LIN {X 0,Y 256.069,Z 339.565,A -85,B 0,C 180,E1 -18517.403,E2 -18517.403} C_VEL
LIN {X 0,Y 256.173,Z 339.546,A -85,B 0,C 180,E1 -18520.779,E2 -18520.779} C_VEL
LIN {X 0,Y 256.276,Z 339.562,A -85,B 0,C 180,E1 -18524.084,E2 -18524.084} C_VEL
LIN {X 0,Y 256.286,Z 339.555,A -85,B 0,C 180,E1 -18528.933,E2 -18528.933} C_VEL
LIN {X 0,Y 256.491,Z 339.526,A -85,B 0,C 180,E1 -18532.126,E2 -18532.126} C_VEL
LIN {X 0,Y 256.447,Z 339.54,A -85,B 0,C 180,E1 -18536.858,E2 -18536.858} C_VEL
LIN {X 0,Y 256.694,Z 339.506,A -85,B 0,C 180,E1 -18538.431,E2 -18538.431} C_VEL
LIN {X 0,Y 256.692,Z 339.489,A -85,B 0,C 180,E1 -18541.569,E2 -18541.569} C_VEL
LIN {X 0,Y 256.437,Z 339.527,A -85,B 0,C 180,E1 -18546.594,E2 -18546.594} C_VEL
LIN {X 0,Y 256.423,Z 339.532,A -85,B 0,C 180,E1 -18549.465,E2 -18549.465} C_VEL
LIN {X 0,Y 256.231,Z 339.545,A -85,B 0,C 180,E1 -18554.292,E2 -18554.292} C_VEL
LIN {X 0,Y 256.173,Z 339.575,A -85,B 0,C 180,E1 -18557.565,E2 -18557.565} C_VEL
LIN {X 0,Y 256.133,Z 339.561,A -85,B 0,C 180,E1 -18561.108,E2 -18561.108} C_VEL
LIN {X 0,Y 256.078,Z 339.583,A -85,B 0,C 180,E1 -18565.088,E2 -18565.088} C_VEL
LIN {X 0,Y 256.072,Z 339.529,A -85,B 0,C 180,E1 -18568.57,E2 -18568.57} C_VEL
LIN {X 0,Y 256.066,Z 339.546,A -85,B 0,C 180,E1 -18571.7,E2 -18571.7} C_VEL
LIN {X 0,Y 256.076,Z 339.588,A -85,B 0,C 180,E1 -18575.194,E2 -18575.194} C_VEL
LIN {X 0,Y 256.062,Z 339.542,A -85,B 0,C 180,E1 -18579.144,E2 -18579.144} C_VEL
LIN {X 0,Y 256.02,Z 339.597,A -85,B 0,C 180,E1 -18583.336,E2 -18583.336} C_VEL
LIN {X 0,Y 256.031,Z 339.564,A -85,B 0,C 180,E1 -18587.829,E2 -18587.829} C_VEL
LIN {X 0,Y 256.064,Z 339.581,A -85,B 0,C 180,E1 -18590.857,E2 -18590.857} C_VEL
LIN {X 0,Y 256.078,Z 339.583,A -85,B 0,C 180,E1 -18594.807,E2 -18594.807} C_VEL
LIN {X 0,Y 256.112,Z 339.714,A -85,B 0,C 180,E1 -18598.125,E2 -18598.125} C_VEL
LIN {X 0,Y 256.299,Z 340.625,A -85,B 0,C 180,E1 -18598.413,E2 -18598.413} C_VEL
LIN {X 0,Y 265.977,Z 358.451,A -85,B 0,C 180,E1 -18600.315,E2 -18600.315} C_VEL
LIN {X 0,Y 273.395,Z 374.129,A -85,B 0,C 180,E1 -18601.697,E2 -18601.697} C_VEL
LIN {X 0,Y 273.811,Z 374.994,A -85,B 0,C 180,E1 -18601.771,E2 -18601.771} C_VEL
LIN {X 0,Y 272.891,Z 418.973,A -85,B 0,C 180,E1 -18602.963,E2 -18602.963} C_VEL
LIN {X 0,Y 272.46,Z 432.928,A -85,B 0,C 180,E1 -18603.563,E2 -18603.563} C_VEL
LIN {X 0,Y 271.747,Z 444.5,A -85,B 0,C 180,E1 -18604.331,E2 -18604.331} C_VEL
LIN {X 0,Y 270.545,Z 456.738,A -85,B 0,C 180,E1 -18605.441,E2 -18605.441} C_VEL
LIN {X 0,Y 269.175,Z 467,A -85,B 0,C 180,E1 -18606.638,E2 -18606.638} C_VEL
LIN {X 0,Y 267.356,Z 477.747,A -85,B 0,C 180,E1 -18608.204,E2 -18608.204} C_VEL
LIN {X 0,Y 265.658,Z 486.939,A -85,B 0,C 180,E1 -18609.885,E2 -18609.885} C_VEL
LIN {X 0,Y 264.051,Z 495.288,A -85,B 0,C 180,E1 -18611.776,E2 -18611.776} C_VEL
LIN {X 0,Y 262.199,Z 503.403,A -85,B 0,C 180,E1 -18614.054,E2 -18614.054} C_VEL
LIN {X 0,Y 260.462,Z 510.51,A -85,B 0,C 180,E1 -18616.578,E2 -18616.578} C_VEL
LIN {X 0,Y 259.237,Z 515.882,A -85,B 0,C 180,E1 -18619.061,E2 -18619.061} C_VEL
LIN {X 0,Y 258.088,Z 519.772,A -85,B 0,C 180,E1 -18621.387,E2 -18621.387} C_VEL
LIN {X 0,Y 257.177,Z 522.649,A -85,B 0,C 180,E1 -18623.725,E2 -18623.725} C_VEL
LIN {X 0,Y 257.015,Z 523.987,A -85,B 0,C 180,E1 -18625.295,E2 -18625.295} C_VEL
LIN {X 0,Y 256.72,Z 524.962,A -85,B 0,C 180,E1 -18626.861,E2 -18626.861} C_VEL
LIN {X 0,Y 256.704,Z 525.54,A -85,B 0,C 180,E1 -18628.431,E2 -18628.431} C_VEL
LIN {X 0,Y 256.664,Z 525.764,A -85,B 0,C 180,E1 -18630,E2 -18630} C_VEL
LIN {X 0,Y 256.704,Z 525.576,A -85,B 0,C 180,E1 -18631.569,E2 -18631.569} C_VEL
LIN {X 0,Y 256.719,Z 525.022,A -85,B 0,C 180,E1 -18633.139,E2 -18633.139} C_VEL
LIN {X 0,Y 257.009,Z 524.07,A -85,B 0,C 180,E1 -18634.706,E2 -18634.706} C_VEL
LIN {X 0,Y 257.163,Z 522.771,A -85,B 0,C 180,E1 -18636.276,E2 -18636.276} C_VEL
LIN {X 0,Y 258.081,Z 519.939,A -85,B 0,C 180,E1 -18638.614,E2 -18638.614} C_VEL
LIN {X 0,Y 259.211,Z 516.108,A -85,B 0,C 180,E1 -18640.94,E2 -18640.94} C_VEL
LIN {X 0,Y 260.376,Z 511.024,A -85,B 0,C 180,E1 -18643.342,E2 -18643.342} C_VEL
LIN {X 0,Y 262.21,Z 503.778,A -85,B 0,C 180,E1 -18645.946,E2 -18645.946} C_VEL
LIN {X 0,Y 264.037,Z 495.746,A -85,B 0,C 180,E1 -18648.225,E2 -18648.225} C_VEL
LIN {X 0,Y 265.659,Z 487.519,A -85,B 0,C 180,E1 -18650.115,E2 -18650.115} C_VEL
LIN {X 0,Y 267.297,Z 478.476,A -85,B 0,C 180,E1 -18651.801,E2 -18651.801} C_VEL
LIN {X 0,Y 269.348,Z 466.924,A -85,B 0,C 180,E1 -18653.483,E2 -18653.483} C_VEL
LIN {X 0,Y 270.868,Z 454.986,A -85,B 0,C 180,E1 -18654.859,E2 -18654.859} C_VEL
LIN {X 0,Y 272.101,Z 442.376,A -85,B 0,C 180,E1 -18655.932,E2 -18655.932} C_VEL
LIN {X 0,Y 272.774,Z 430.266,A -85,B 0,C 180,E1 -18656.684,E2 -18656.684} C_VEL
LIN {X 0,Y 272.92,Z 419.568,A -85,B 0,C 180,E1 -18657.142,E2 -18657.142} C_VEL
LIN {X 0,Y 273.881,Z 375.117,A -85,B 0,C 180,E1 -18658.347,E2 -18658.347} C_VEL
LIN {X 0,Y 266.772,Z 359.974,A -85,B 0,C 180,E1 -18659.671,E2 -18659.671} C_VEL
LIN {X 0,Y 259.254,Z 346.14,A -85,B 0,C 180,E1 -18661.101,E2 -18661.101} C_VEL
LIN {X 0,Y 256.306,Z 340.687,A -85,B 0,C 180,E1 -18661.719,E2 -18661.719} C_VEL
LIN {X 0,Y 256.095,Z 339.689,A -85,B 0,C 180,E1 -18662.04,E2 -18662.04} C_VEL
LIN {X 0,Y 256.077,Z 339.586,A -85,B 0,C 180,E1 -18665.193,E2 -18665.193} C_VEL
LIN {X 0,Y 256.041,Z 339.582,A -85,B 0,C 180,E1 -18669.147,E2 -18669.147} C_VEL
LIN {X 0,Y 256.001,Z 339.563,A -85,B 0,C 180,E1 -18673.339,E2 -18673.339} C_VEL
LIN {X 0,Y 256.031,Z 339.586,A -85,B 0,C 180,E1 -18677.828,E2 -18677.828} C_VEL
LIN {X 0,Y 256.062,Z 339.543,A -85,B 0,C 180,E1 -18680.856,E2 -18680.856} C_VEL
LIN {X 0,Y 256.076,Z 339.587,A -85,B 0,C 180,E1 -18684.806,E2 -18684.806} C_VEL
LIN {X 0,Y 256.074,Z 339.541,A -85,B 0,C 180,E1 -18688.57,E2 -18688.57} C_VEL
LIN {X 0,Y 256.073,Z 339.538,A -85,B 0,C 180,E1 -18692.188,E2 -18692.188} C_VEL
LIN {X 0,Y 256.081,Z 339.586,A -85,B 0,C 180,E1 -18695.69,E2 -18695.69} C_VEL
LIN {X 0,Y 256.117,Z 339.563,A -85,B 0,C 180,E1 -18699.1,E2 -18699.1} C_VEL
LIN {X 0,Y 256.226,Z 339.555,A -85,B 0,C 180,E1 -18704.08,E2 -18704.08} C_VEL
LIN {X 0,Y 256.286,Z 339.56,A -85,B 0,C 180,E1 -18708.933,E2 -18708.933} C_VEL
LIN {X 0,Y 256.462,Z 339.518,A -85,B 0,C 180,E1 -18712.125,E2 -18712.125} C_VEL
LIN {X 0,Y 256.449,Z 339.535,A -85,B 0,C 180,E1 -18716.858,E2 -18716.858} C_VEL
LIN {X 0,Y 256.691,Z 339.489,A -85,B 0,C 180,E1 -18718.431,E2 -18718.431} C_VEL
LIN {X 0,Y 256.637,Z 339.511,A -85,B 0,C 180,E1 -18721.842,E2 -18721.842} C_VEL
LIN {X 0,Y 256.452,Z 339.518,A -85,B 0,C 180,E1 -18726.293,E2 -18726.293} C_VEL
LIN {X 0,Y 256.424,Z 339.535,A -85,B 0,C 180,E1 -18728.703,E2 -18728.703} C_VEL
LIN {X 0,Y 255.723,Z 339.631,A -85,B 0,C 180,E1 -18730.013,E2 -18730.013} C_VEL
LIN {X 0,Y 252.772,Z 339.993,A -85,B 0,C 180,E1 -18732.144,E2 -18732.144} C_VEL
LIN {X 0,Y 250.284,Z 340.298,A -85,B 0,C 180,E1 -18733.88,E2 -18733.88} C_VEL
LIN {X 0,Y 249.236,Z 340.437,A -85,B 0,C 180,E1 -18735.229,E2 -18735.229} C_VEL
LIN {X 0,Y 249.16,Z 340.442,A -85,B 0,C 180,E1 -18735.686,E2 -18735.686} C_VEL
LIN {X 0,Y 249.08,Z 340.421,A -85,B 0,C 180,E1 -18739.791,E2 -18739.791} C_VEL
LIN {X 0,Y 249.039,Z 340.452,A -85,B 0,C 180,E1 -18743.271,E2 -18743.271} C_VEL
LIN {X 0,Y 249.02,Z 340.448,A -85,B 0,C 180,E1 -18746.844,E2 -18746.844} C_VEL
LIN {X 0,Y 248.998,Z 340.46,A -85,B 0,C 180,E1 -18750.534,E2 -18750.534} C_VEL
LIN {X 0,Y 249.04,Z 340.444,A -85,B 0,C 180,E1 -18755.077,E2 -18755.077} C_VEL
LIN {X 0,Y 249.02,Z 340.455,A -85,B 0,C 180,E1 -18758.382,E2 -18758.382} C_VEL
LIN {X 0,Y 248.98,Z 340.447,A -85,B 0,C 180,E1 -18762.786,E2 -18762.786} C_VEL
LIN {X 0,Y 248.985,Z 340.61,A -85,B 0,C 180,E1 -18765.118,E2 -18765.118} C_VEL
LIN {X 0,Y 252.25,Z 352.179,A -85,B 0,C 180,E1 -18769.37,E2 -18769.37} C_VEL
LIN {X 0,Y 254.64,Z 361.802,A -85,B 0,C 180,E1 -18772.614,E2 -18772.614} C_VEL
LIN {X 0,Y 256.671,Z 371.259,A -85,B 0,C 180,E1 -18775.613,E2 -18775.613} C_VEL
LIN {X 0,Y 257.459,Z 376.644,A -85,B 0,C 180,E1 -18777.232,E2 -18777.232} C_VEL
LIN {X 0,Y 257.14,Z 378.887,A -85,B 0,C 180,E1 -18777.719,E2 -18777.719} C_VEL
LIN {X 0,Y 260.773,Z 406.312,A -85,B 0,C 180,E1 -18779.087,E2 -18779.087} C_VEL
LIN {X 0,Y 263.817,Z 435.444,A -85,B 0,C 180,E1 -18780.357,E2 -18780.357} C_VEL
LIN {X 0,Y 265.192,Z 455.664,A -85,B 0,C 180,E1 -18781.128,E2 -18781.128} C_VEL
LIN {X 0,Y 263.991,Z 490.905,A -85,B 0,C 180,E1 -18782.108,E2 -18782.108} C_VEL
LIN {X 0,Y 262.825,Z 504.718,A -85,B 0,C 180,E1 -18782.791,E2 -18782.791} C_VEL
LIN {X 0,Y 261.078,Z 517.612,A -85,B 0,C 180,E1 -18783.738,E2 -18783.738} C_VEL
LIN {X 0,Y 259.146,Z 529.368,A -85,B 0,C 180,E1 -18784.929,E2 -18784.929} C_VEL
LIN {X 0,Y 256.812,Z 540.726,A -85,B 0,C 180,E1 -18786.408,E2 -18786.408} C_VEL
LIN {X 0,Y 254.578,Z 551.008,A -85,B 0,C 180,E1 -18788.119,E2 -18788.119} C_VEL
LIN {X 0,Y 252.455,Z 560.299,A -85,B 0,C 180,E1 -18790.061,E2 -18790.061} C_VEL
LIN {X 0,Y 250.616,Z 569.039,A -85,B 0,C 180,E1 -18792.34,E2 -18792.34} C_VEL
LIN {X 0,Y 249.503,Z 574.497,A -85,B 0,C 180,E1 -18794.06,E2 -18794.06} C_VEL
LIN {X 0,Y 248.311,Z 581.828,A -85,B 0,C 180,E1 -18796.914,E2 -18796.914} C_VEL
LIN {X 0,Y 247.795,Z 586.756,A -85,B 0,C 180,E1 -18799.377,E2 -18799.377} C_VEL
LIN {X 0,Y 247.778,Z 590.581,A -85,B 0,C 180,E1 -18801.847,E2 -18801.847} C_VEL
LIN {X 0,Y 247.949,Z 592.578,A -85,B 0,C 180,E1 -18803.49,E2 -18803.49} C_VEL
LIN {X 0,Y 248.237,Z 594.099,A -85,B 0,C 180,E1 -18805.128,E2 -18805.128} C_VEL
LIN {X 0,Y 248.493,Z 595.191,A -85,B 0,C 180,E1 -18806.757,E2 -18806.757} C_VEL
LIN {X 0,Y 248.804,Z 595.878,A -85,B 0,C 180,E1 -18808.381,E2 -18808.381} C_VEL
LIN {X 0,Y 249.239,Z 596.163,A -85,B 0,C 180,E1 -18810,E2 -18810} C_VEL
LIN {X 0,Y 248.809,Z 595.869,A -85,B 0,C 180,E1 -18811.619,E2 -18811.619} C_VEL
LIN {X 0,Y 248.504,Z 595.178,A -85,B 0,C 180,E1 -18813.242,E2 -18813.242} C_VEL
LIN {X 0,Y 248.257,Z 594.082,A -85,B 0,C 180,E1 -18814.872,E2 -18814.872} C_VEL
LIN {X 0,Y 247.899,Z 591.823,A -85,B 0,C 180,E1 -18817.132,E2 -18817.132} C_VEL
LIN {X 0,Y 247.761,Z 588.091,A -85,B 0,C 180,E1 -18819.799,E2 -18819.799} C_VEL
LIN {X 0,Y 248.096,Z 583.525,A -85,B 0,C 180,E1 -18822.266,E2 -18822.266} C_VEL
LIN {X 0,Y 248.876,Z 577.769,A -85,B 0,C 180,E1 -18824.723,E2 -18824.723} C_VEL
LIN {X 0,Y 249.858,Z 571.762,A -85,B 0,C 180,E1 -18826.805,E2 -18826.805} C_VEL
LIN {X 0,Y 251.413,Z 564.965,A -85,B 0,C 180,E1 -18828.752,E2 -18828.752} C_VEL
LIN {X 0,Y 253.248,Z 556.625,A -85,B 0,C 180,E1 -18830.721,E2 -18830.721} C_VEL
LIN {X 0,Y 255.584,Z 546.518,A -85,B 0,C 180,E1 -18832.641,E2 -18832.641} C_VEL
LIN {X 0,Y 257.668,Z 536.556,A -85,B 0,C 180,E1 -18834.15,E2 -18834.15} C_VEL
LIN {X 0,Y 260.045,Z 523.989,A -85,B 0,C 180,E1 -18835.621,E2 -18835.621} C_VEL
LIN {X 0,Y 261.894,Z 511.65,A -85,B 0,C 180,E1 -18836.71,E2 -18836.71} C_VEL
LIN {X 0,Y 263.306,Z 498.554,A -85,B 0,C 180,E1 -18837.526,E2 -18837.526} C_VEL
LIN {X 0,Y 264.182,Z 485.189,A -85,B 0,C 180,E1 -18838.054,E2 -18838.054} C_VEL
LIN {X 0,Y 265.101,Z 453.13,A -85,B 0,C 180,E1 -18838.919,E2 -18838.919} C_VEL
LIN {X 0,Y 262.594,Z 423.589,A -85,B 0,C 180,E1 -18840.111,E2 -18840.111} C_VEL
LIN {X 0,Y 259.354,Z 395.566,A -85,B 0,C 180,E1 -18841.387,E2 -18841.387} C_VEL
LIN {X 0,Y 257.067,Z 378.809,A -85,B 0,C 180,E1 -18842.247,E2 -18842.247} C_VEL
LIN {X 0,Y 257.402,Z 375.362,A -85,B 0,C 180,E1 -18843.097,E2 -18843.097} C_VEL
LIN {X 0,Y 255.441,Z 365.273,A -85,B 0,C 180,E1 -18846.216,E2 -18846.216} C_VEL
LIN {X 0,Y 252.585,Z 353.374,A -85,B 0,C 180,E1 -18850.154,E2 -18850.154} C_VEL
LIN {X 0,Y 249.584,Z 342.552,A -85,B 0,C 180,E1 -18854.06,E2 -18854.06} C_VEL
LIN {X 0,Y 248.977,Z 340.558,A -85,B 0,C 180,E1 -18854.884,E2 -18854.884} C_VEL
LIN {X 0,Y 248.99,Z 340.452,A -85,B 0,C 180,E1 -18857.357,E2 -18857.357} C_VEL
LIN {X 0,Y 249.04,Z 340.389,A -85,B 0,C 180,E1 -18862.2,E2 -18862.2} C_VEL
LIN {X 0,Y 249.039,Z 340.419,A -85,B 0,C 180,E1 -18865.639,E2 -18865.639} C_VEL
LIN {X 0,Y 248.998,Z 340.459,A -85,B 0,C 180,E1 -18869.466,E2 -18869.466} C_VEL
LIN {X 0,Y 249.02,Z 340.45,A -85,B 0,C 180,E1 -18873.156,E2 -18873.156} C_VEL
LIN {X 0,Y 249.04,Z 340.451,A -85,B 0,C 180,E1 -18876.729,E2 -18876.729} C_VEL
LIN {X 0,Y 249.094,Z 340.42,A -85,B 0,C 180,E1 -18880.21,E2 -18880.21} C_VEL
LIN {X 0,Y 249.22,Z 340.442,A -85,B 0,C 180,E1 -18883.62,E2 -18883.62} C_VEL
LIN {X 0,Y 249.23,Z 340.43,A -85,B 0,C 180,E1 -18888.616,E2 -18888.616} C_VEL
LIN {X 0,Y 249.434,Z 340.406,A -85,B 0,C 180,E1 -18891.901,E2 -18891.901} C_VEL
LIN {X 0,Y 249.259,Z 340.423,A -85,B 0,C 180,E1 -18895.148,E2 -18895.148} C_VEL
LIN {X 0,Y 249.655,Z 340.383,A -85,B 0,C 180,E1 -18898.387,E2 -18898.387} C_VEL
LIN {X 0,Y 249.653,Z 340.366,A -85,B 0,C 180,E1 -18901.613,E2 -18901.613} C_VEL
LIN {X 0,Y 249.414,Z 340.401,A -85,B 0,C 180,E1 -18906.573,E2 -18906.573} C_VEL
LIN {X 0,Y 249.339,Z 340.416,A -85,B 0,C 180,E1 -18909.737,E2 -18909.737} C_VEL
LIN {X 0,Y 249.174,Z 340.423,A -85,B 0,C 180,E1 -18914.705,E2 -18914.705} C_VEL
LIN {X 0,Y 249.108,Z 340.454,A -85,B 0,C 180,E1 -18918.08,E2 -18918.08} C_VEL
LIN {X 0,Y 249.073,Z 340.441,A -85,B 0,C 180,E1 -18921.52,E2 -18921.52} C_VEL
LIN {X 0,Y 249.039,Z 340.455,A -85,B 0,C 180,E1 -18925.44,E2 -18925.44} C_VEL
LIN {X 0,Y 249.02,Z 340.403,A -85,B 0,C 180,E1 -18928.969,E2 -18928.969} C_VEL
LIN {X 0,Y 249.022,Z 340.438,A -85,B 0,C 180,E1 -18932.427,E2 -18932.427} C_VEL
LIN {X 0,Y 249.01,Z 340.454,A -85,B 0,C 180,E1 -18936.349,E2 -18936.349} C_VEL
LIN {X 0,Y 248.976,Z 340.432,A -85,B 0,C 180,E1 -18940.484,E2 -18940.484} C_VEL
LIN {X 0,Y 248.96,Z 340.457,A -85,B 0,C 180,E1 -18944.889,E2 -18944.889} C_VEL
LIN {X 0,Y 248.977,Z 340.438,A -85,B 0,C 180,E1 -18947.355,E2 -18947.355} C_VEL
LIN {X 0,Y 249.017,Z 340.447,A -85,B 0,C 180,E1 -18951.619,E2 -18951.619} C_VEL
LIN {X 0,Y 249.042,Z 340.46,A -85,B 0,C 180,E1 -18955.64,E2 -18955.64} C_VEL
LIN {X 0,Y 249.084,Z 340.699,A -85,B 0,C 180,E1 -18957.164,E2 -18957.164} C_VEL
LIN {X 0,Y 249.404,Z 341.93,A -85,B 0,C 180,E1 -18957.457,E2 -18957.457} C_VEL
LIN {X 0,Y 258.456,Z 358.147,A -85,B 0,C 180,E1 -18959.31,E2 -18959.31} C_VEL
LIN {X 0,Y 265.998,Z 373.461,A -85,B 0,C 180,E1 -18960.778,E2 -18960.778} C_VEL
LIN {X 0,Y 267.575,Z 377.081,A -85,B 0,C 180,E1 -18961.084,E2 -18961.084} C_VEL
LIN {X 0,Y 266.644,Z 419.863,A -85,B 0,C 180,E1 -18962.272,E2 -18962.272} C_VEL
LIN {X 0,Y 266.201,Z 433.521,A -85,B 0,C 180,E1 -18962.868,E2 -18962.868} C_VEL
LIN {X 0,Y 265.425,Z 445.487,A -85,B 0,C 180,E1 -18963.673,E2 -18963.673} C_VEL
LIN {X 0,Y 264.169,Z 457.722,A -85,B 0,C 180,E1 -18964.808,E2 -18964.808} C_VEL
LIN {X 0,Y 262.738,Z 467.983,A -85,B 0,C 180,E1 -18966.03,E2 -18966.03} C_VEL
LIN {X 0,Y 260.844,Z 478.729,A -85,B 0,C 180,E1 -18967.631,E2 -18967.631} C_VEL
LIN {X 0,Y 259.069,Z 487.921,A -85,B 0,C 180,E1 -18969.35,E2 -18969.35} C_VEL
LIN {X 0,Y 257.384,Z 496.268,A -85,B 0,C 180,E1 -18971.287,E2 -18971.287} C_VEL
LIN {X 0,Y 255.448,Z 504.383,A -85,B 0,C 180,E1 -18973.621,E2 -18973.621} C_VEL
LIN {X 0,Y 253.631,Z 511.49,A -85,B 0,C 180,E1 -18976.21,E2 -18976.21} C_VEL
LIN {X 0,Y 252.34,Z 516.861,A -85,B 0,C 180,E1 -18978.758,E2 -18978.758} C_VEL
LIN {X 0,Y 251.142,Z 520.751,A -85,B 0,C 180,E1 -18981.146,E2 -18981.146} C_VEL
LIN {X 0,Y 250.189,Z 523.628,A -85,B 0,C 180,E1 -18983.549,E2 -18983.549} C_VEL
LIN {X 0,Y 250.01,Z 524.965,A -85,B 0,C 180,E1 -18985.162,E2 -18985.162} C_VEL
LIN {X 0,Y 249.703,Z 525.94,A -85,B 0,C 180,E1 -18986.773,E2 -18986.773} C_VEL
LIN {X 0,Y 249.679,Z 526.518,A -85,B 0,C 180,E1 -18988.387,E2 -18988.387} C_VEL
LIN {X 0,Y 249.636,Z 526.742,A -85,B 0,C 180,E1 -18990,E2 -18990} C_VEL
LIN {X 0,Y 249.679,Z 526.554,A -85,B 0,C 180,E1 -18991.613,E2 -18991.613} C_VEL
LIN {X 0,Y 249.702,Z 525.999,A -85,B 0,C 180,E1 -18993.227,E2 -18993.227} C_VEL
LIN {X 0,Y 250.004,Z 525.048,A -85,B 0,C 180,E1 -18994.838,E2 -18994.838} C_VEL
LIN {X 0,Y 250.174,Z 523.749,A -85,B 0,C 180,E1 -18996.452,E2 -18996.452} C_VEL
LIN {X 0,Y 251.135,Z 520.916,A -85,B 0,C 180,E1 -18998.854,E2 -18998.854} C_VEL
LIN {X 0,Y 252.315,Z 517.085,A -85,B 0,C 180,E1 -19001.243,E2 -19001.243} C_VEL
LIN {X 0,Y 253.543,Z 512,A -85,B 0,C 180,E1 -19003.709,E2 -19003.709} C_VEL
LIN {X 0,Y 255.459,Z 504.754,A -85,B 0,C 180,E1 -19006.379,E2 -19006.379} C_VEL
LIN {X 0,Y 257.371,Z 496.722,A -85,B 0,C 180,E1 -19008.714,E2 -19008.714} C_VEL
LIN {X 0,Y 259.069,Z 488.494,A -85,B 0,C 180,E1 -19010.65,E2 -19010.65} C_VEL
LIN {X 0,Y 260.785,Z 479.451,A -85,B 0,C 180,E1 -19012.374,E2 -19012.374} C_VEL
LIN {X 0,Y 262.729,Z 468.921,A -85,B 0,C 180,E1 -19013.96,E2 -19013.96} C_VEL
LIN {X 0,Y 264.342,Z 457.235,A -85,B 0,C 180,E1 -19015.364,E2 -19015.364} C_VEL
LIN {X 0,Y 265.643,Z 445.757,A -85,B 0,C 180,E1 -19016.41,E2 -19016.41} C_VEL
LIN {X 0,Y 266.365,Z 433.594,A -85,B 0,C 180,E1 -19017.241,E2 -19017.241} C_VEL
LIN {X 0,Y 266.676,Z 420.237,A -85,B 0,C 180,E1 -19017.843,E2 -19017.843} C_VEL
LIN {X 0,Y 267.652,Z 377.15,A -85,B 0,C 180,E1 -19019.037,E2 -19019.037} C_VEL
LIN {X 0,Y 260.711,Z 362.373,A -85,B 0,C 180,E1 -19020.387,E2 -19020.387} C_VEL
LIN {X 0,Y 252.472,Z 347.365,A -85,B 0,C 180,E1 -19022.029,E2 -19022.029} C_VEL
LIN {X 0,Y 249.294,Z 341.581,A -85,B 0,C 180,E1 -19022.729,E2 -19022.729} C_VEL
LIN {X 0,Y 249.048,Z 340.566,A -85,B 0,C 180,E1 -19023.087,E2 -19023.087} C_VEL
LIN {X 0,Y 249.01,Z 340.448,A -85,B 0,C 180,E1 -19026.348,E2 -19026.348} C_VEL
LIN {X 0,Y 248.97,Z 340.471,A -85,B 0,C 180,E1 -19030.484,E2 -19030.484} C_VEL
LIN {X 0,Y 248.96,Z 340.452,A -85,B 0,C 180,E1 -19034.888,E2 -19034.888} C_VEL
LIN {X 0,Y 248.977,Z 340.472,A -85,B 0,C 180,E1 -19037.354,E2 -19037.354} C_VEL
LIN {X 0,Y 249.041,Z 340.424,A -85,B 0,C 180,E1 -19042.2,E2 -19042.2} C_VEL
LIN {X 0,Y 249.04,Z 340.463,A -85,B 0,C 180,E1 -19045.639,E2 -19045.639} C_VEL
LIN {X 0,Y 248.99,Z 340.409,A -85,B 0,C 180,E1 -19049.464,E2 -19049.464} C_VEL
LIN {X 0,Y 249.009,Z 340.436,A -85,B 0,C 180,E1 -19053.155,E2 -19053.155} C_VEL
LIN {X 0,Y 249.002,Z 340.466,A -85,B 0,C 180,E1 -19056.725,E2 -19056.725} C_VEL
LIN {X 0,Y 249.052,Z 340.449,A -85,B 0,C 180,E1 -19060.207,E2 -19060.207} C_VEL
LIN {X 0,Y 249.154,Z 340.442,A -85,B 0,C 180,E1 -19063.616,E2 -19063.616} C_VEL
LIN {X 0,Y 249.229,Z 340.441,A -85,B 0,C 180,E1 -19068.615,E2 -19068.615} C_VEL
LIN {X 0,Y 249.412,Z 340.396,A -85,B 0,C 180,E1 -19071.9,E2 -19071.9} C_VEL
LIN {X 0,Y 249.26,Z 340.436,A -85,B 0,C 180,E1 -19075.148,E2 -19075.148} C_VEL
LIN {X 0,Y 249.653,Z 340.366,A -85,B 0,C 180,E1 -19078.387,E2 -19078.387} C_VEL
LIN {X 0,Y 249.655,Z 340.382,A -85,B 0,C 180,E1 -19081.613,E2 -19081.613} C_VEL
LIN {X 0,Y 249.423,Z 340.394,A -85,B 0,C 180,E1 -19086.471,E2 -19086.471} C_VEL
LIN {X 0,Y 249.339,Z 340.425,A -85,B 0,C 180,E1 -19089.737,E2 -19089.737} C_VEL
LIN {X 0,Y 249.177,Z 340.439,A -85,B 0,C 180,E1 -19094.705,E2 -19094.705} C_VEL
LIN {X 0,Y 249.16,Z 340.442,A -85,B 0,C 180,E1 -19095.686,E2 -19095.686} C_VEL
LIN {X 0,Y 248.504,Z 340.527,A -85,B 0,C 180,E1 -19097.035,E2 -19097.035} C_VEL
LIN {X 0,Y 245.605,Z 340.872,A -85,B 0,C 180,E1 -19099.233,E2 -19099.233} C_VEL
LIN {X 0,Y 243.125,Z 341.169,A -85,B 0,C 180,E1 -19101.023,E2 -19101.023} C_VEL
LIN {X 0,Y 242.058,Z 341.307,A -85,B 0,C 180,E1 -19102.414,E2 -19102.414} C_VEL
LIN {X 0,Y 241.971,Z 341.321,A -85,B 0,C 180,E1 -19102.886,E2 -19102.886} C_VEL
LIN {X 0,Y 241.988,Z 341.337,A -85,B 0,C 180,E1 -19105.826,E2 -19105.826} C_VEL
LIN {X 0,Y 241.965,Z 341.322,A -85,B 0,C 180,E1 -19109.589,E2 -19109.589} C_VEL
LIN {X 0,Y 241.976,Z 341.327,A -85,B 0,C 180,E1 -19113.493,E2 -19113.493} C_VEL
LIN {X 0,Y 241.981,Z 341.341,A -85,B 0,C 180,E1 -19117.584,E2 -19117.584} C_VEL
LIN {X 0,Y 241.915,Z 341.346,A -85,B 0,C 180,E1 -19121.927,E2 -19121.927} C_VEL
LIN {X 0,Y 241.93,Z 341.545,A -85,B 0,C 180,E1 -19124.202,E2 -19124.202} C_VEL
LIN {X 0,Y 244.942,Z 352.046,A -85,B 0,C 180,E1 -19128.246,E2 -19128.246} C_VEL
LIN {X 0,Y 247.415,Z 361.774,A -85,B 0,C 180,E1 -19131.687,E2 -19131.687} C_VEL
LIN {X 0,Y 249.909,Z 373.223,A -85,B 0,C 180,E1 -19135.462,E2 -19135.462} C_VEL
LIN {X 0,Y 250.67,Z 377.47,A -85,B 0,C 180,E1 -19136.741,E2 -19136.741} C_VEL
LIN {X 0,Y 252.007,Z 387.42,A -85,B 0,C 180,E1 -19137.314,E2 -19137.314} C_VEL
LIN {X 0,Y 254.816,Z 408.963,A -85,B 0,C 180,E1 -19138.397,E2 -19138.397} C_VEL
LIN {X 0,Y 257.963,Z 440.471,A -85,B 0,C 180,E1 -19139.8,E2 -19139.8} C_VEL
LIN {X 0,Y 258.942,Z 455.77,A -85,B 0,C 180,E1 -19140.396,E2 -19140.396} C_VEL
LIN {X 0,Y 257.731,Z 489.933,A -85,B 0,C 180,E1 -19141.369,E2 -19141.369} C_VEL
LIN {X 0,Y 256.53,Z 503.249,A -85,B 0,C 180,E1 -19142.031,E2 -19142.031} C_VEL
LIN {X 0,Y 254.926,Z 515.618,A -85,B 0,C 180,E1 -19142.943,E2 -19142.943} C_VEL
LIN {X 0,Y 253.049,Z 526.794,A -85,B 0,C 180,E1 -19144.06,E2 -19144.06} C_VEL
LIN {X 0,Y 250.607,Z 538.439,A -85,B 0,C 180,E1 -19145.566,E2 -19145.566} C_VEL
LIN {X 0,Y 248.198,Z 548.961,A -85,B 0,C 180,E1 -19147.307,E2 -19147.307} C_VEL
LIN {X 0,Y 246.186,Z 557.607,A -85,B 0,C 180,E1 -19149.094,E2 -19149.094} C_VEL
LIN {X 0,Y 244.331,Z 565.623,A -85,B 0,C 180,E1 -19151.12,E2 -19151.12} C_VEL
LIN {X 0,Y 242.537,Z 573.489,A -85,B 0,C 180,E1 -19153.589,E2 -19153.589} C_VEL
LIN {X 0,Y 241.339,Z 580.832,A -85,B 0,C 180,E1 -19156.528,E2 -19156.528} C_VEL
LIN {X 0,Y 240.763,Z 585.761,A -85,B 0,C 180,E1 -19159.063,E2 -19159.063} C_VEL
LIN {X 0,Y 240.708,Z 589.587,A -85,B 0,C 180,E1 -19161.606,E2 -19161.606} C_VEL
LIN {X 0,Y 240.856,Z 591.585,A -85,B 0,C 180,E1 -19163.297,E2 -19163.297} C_VEL
LIN {X 0,Y 241.145,Z 593.109,A -85,B 0,C 180,E1 -19164.984,E2 -19164.984} C_VEL
LIN {X 0,Y 241.432,Z 594.207,A -85,B 0,C 180,E1 -19166.662,E2 -19166.662} C_VEL
LIN {X 0,Y 241.741,Z 594.895,A -85,B 0,C 180,E1 -19168.334,E2 -19168.334} C_VEL
LIN {X 0,Y 242.198,Z 595.183,A -85,B 0,C 180,E1 -19170,E2 -19170} C_VEL
LIN {X 0,Y 241.443,Z 594.194,A -85,B 0,C 180,E1 -19173.337,E2 -19173.337} C_VEL
LIN {X 0,Y 241.166,Z 593.091,A -85,B 0,C 180,E1 -19175.015,E2 -19175.015} C_VEL
LIN {X 0,Y 240.823,Z 591.053,A -85,B 0,C 180,E1 -19177.146,E2 -19177.146} C_VEL
LIN {X 0,Y 240.686,Z 587.091,A -85,B 0,C 180,E1 -19180.09,E2 -19180.09} C_VEL
LIN {X 0,Y 241.087,Z 582.525,A -85,B 0,C 180,E1 -19182.629,E2 -19182.629} C_VEL
LIN {X 0,Y 241.954,Z 576.771,A -85,B 0,C 180,E1 -19185.154,E2 -19185.154} C_VEL
LIN {X 0,Y 242.857,Z 571.45,A -85,B 0,C 180,E1 -19187.069,E2 -19187.069} C_VEL
LIN {X 0,Y 244.631,Z 563.965,A -85,B 0,C 180,E1 -19189.292,E2 -19189.292} C_VEL
LIN {X 0,Y 246.571,Z 555.627,A -85,B 0,C 180,E1 -19191.31,E2 -19191.31} C_VEL
LIN {X 0,Y 248.956,Z 545.513,A -85,B 0,C 180,E1 -19193.279,E2 -19193.279} C_VEL
LIN {X 0,Y 251.479,Z 534.124,A -85,B 0,C 180,E1 -19195.004,E2 -19195.004} C_VEL
LIN {X 0,Y 253.659,Z 522.996,A -85,B 0,C 180,E1 -19196.314,E2 -19196.314} C_VEL
LIN {X 0,Y 255.581,Z 510.656,A -85,B 0,C 180,E1 -19197.425,E2 -19197.425} C_VEL
LIN {X 0,Y 257.023,Z 497.964,A -85,B 0,C 180,E1 -19198.234,E2 -19198.234} C_VEL
LIN {X 0,Y 257.922,Z 484.494,A -85,B 0,C 180,E1 -19198.786,E2 -19198.786} C_VEL
LIN {X 0,Y 258.862,Z 453.924,A -85,B 0,C 180,E1 -19199.628,E2 -19199.628} C_VEL
LIN {X 0,Y 256.159,Z 421.803,A -85,B 0,C 180,E1 -19200.972,E2 -19200.972} C_VEL
LIN {X 0,Y 252.598,Z 391.455,A -85,B 0,C 180,E1 -19202.424,E2 -19202.424} C_VEL
LIN {X 0,Y 250.59,Z 377.511,A -85,B 0,C 180,E1 -19203.216,E2 -19203.216} C_VEL
LIN {X 0,Y 249.442,Z 371.008,A -85,B 0,C 180,E1 -19205.207,E2 -19205.207} C_VEL
LIN {X 0,Y 247.386,Z 361.581,A -85,B 0,C 180,E1 -19208.327,E2 -19208.327} C_VEL
LIN {X 0,Y 244.508,Z 350.507,A -85,B 0,C 180,E1 -19212.256,E2 -19212.256} C_VEL
LIN {X 0,Y 241.923,Z 341.476,A -85,B 0,C 180,E1 -19215.796,E2 -19215.796} C_VEL
LIN {X 0,Y 241.939,Z 341.302,A -85,B 0,C 180,E1 -19220.277,E2 -19220.277} C_VEL
LIN {X 0,Y 241.97,Z 341.276,A -85,B 0,C 180,E1 -19224.486,E2 -19224.486} C_VEL
LIN {X 0,Y 241.95,Z 341.347,A -85,B 0,C 180,E1 -19228.476,E2 -19228.476} C_VEL
LIN {X 0,Y 241.958,Z 341.319,A -85,B 0,C 180,E1 -19232.306,E2 -19232.306} C_VEL
LIN {X 0,Y 242.005,Z 341.336,A -85,B 0,C 180,E1 -19236.01,E2 -19236.01} C_VEL
LIN {X 0,Y 242.025,Z 341.297,A -85,B 0,C 180,E1 -19239.607,E2 -19239.607} C_VEL
LIN {X 0,Y 242.16,Z 341.319,A -85,B 0,C 180,E1 -19243.278,E2 -19243.278} C_VEL
LIN {X 0,Y 242.165,Z 341.305,A -85,B 0,C 180,E1 -19248.279,E2 -19248.279} C_VEL
LIN {X 0,Y 242.384,Z 341.286,A -85,B 0,C 180,E1 -19251.664,E2 -19251.664} C_VEL
LIN {X 0,Y 242.401,Z 341.27,A -85,B 0,C 180,E1 -19253.34,E2 -19253.34} C_VEL
LIN {X 0,Y 242.615,Z 341.26,A -85,B 0,C 180,E1 -19258.34,E2 -19258.34} C_VEL
LIN {X 0,Y 242.613,Z 341.242,A -85,B 0,C 180,E1 -19261.66,E2 -19261.66} C_VEL
LIN {X 0,Y 242.392,Z 341.275,A -85,B 0,C 180,E1 -19266.66,E2 -19266.66} C_VEL
LIN {X 0,Y 242.262,Z 341.301,A -85,B 0,C 180,E1 -19270.024,E2 -19270.024} C_VEL
LIN {X 0,Y 242.132,Z 341.302,A -85,B 0,C 180,E1 -19275.143,E2 -19275.143} C_VEL
LIN {X 0,Y 242.045,Z 341.333,A -85,B 0,C 180,E1 -19278.627,E2 -19278.627} C_VEL
LIN {X 0,Y 241.984,Z 341.33,A -85,B 0,C 180,E1 -19282.183,E2 -19282.183} C_VEL
LIN {X 0,Y 241.983,Z 341.331,A -85,B 0,C 180,E1 -19285.827,E2 -19285.827} C_VEL
LIN {X 0,Y 241.959,Z 341.279,A -85,B 0,C 180,E1 -19289.59,E2 -19289.59} C_VEL
LIN {X 0,Y 241.976,Z 341.335,A -85,B 0,C 180,E1 -19293.494,E2 -19293.494} C_VEL
LIN {X 0,Y 241.98,Z 341.306,A -85,B 0,C 180,E1 -19297.584,E2 -19297.584} C_VEL
LIN {X 0,Y 241.905,Z 341.338,A -85,B 0,C 180,E1 -19301.929,E2 -19301.929} C_VEL
LIN {X 0,Y 241.898,Z 341.318,A -85,B 0,C 180,E1 -19306.581,E2 -19306.581} C_VEL
LIN {X 0,Y 241.988,Z 341.322,A -85,B 0,C 180,E1 -19311.643,E2 -19311.643} C_VEL
LIN {X 0,Y 242.01,Z 341.462,A -85,B 0,C 180,E1 -19315.964,E2 -19315.964} C_VEL
LIN {X 0,Y 242.183,Z 342.274,A -85,B 0,C 180,E1 -19316.297,E2 -19316.297} C_VEL
LIN {X 0,Y 243.705,Z 345.144,A -85,B 0,C 180,E1 -19316.69,E2 -19316.69} C_VEL
LIN {X 0,Y 252.943,Z 361.528,A -85,B 0,C 180,E1 -19318.647,E2 -19318.647} C_VEL
LIN {X 0,Y 260.32,Z 376.615,A -85,B 0,C 180,E1 -19320.146,E2 -19320.146} C_VEL
LIN {X 0,Y 261.393,Z 379.052,A -85,B 0,C 180,E1 -19320.363,E2 -19320.363} C_VEL
LIN {X 0,Y 260.444,Z 420.862,A -85,B 0,C 180,E1 -19321.552,E2 -19321.552} C_VEL
LIN {X 0,Y 259.981,Z 434.173,A -85,B 0,C 180,E1 -19322.143,E2 -19322.143} C_VEL
LIN {X 0,Y 259.142,Z 446.474,A -85,B 0,C 180,E1 -19322.983,E2 -19322.983} C_VEL
LIN {X 0,Y 257.826,Z 458.706,A -85,B 0,C 180,E1 -19324.143,E2 -19324.143} C_VEL
LIN {X 0,Y 256.327,Z 468.969,A -85,B 0,C 180,E1 -19325.392,E2 -19325.392} C_VEL
LIN {X 0,Y 254.359,Z 479.711,A -85,B 0,C 180,E1 -19327.029,E2 -19327.029} C_VEL
LIN {X 0,Y 252.503,Z 488.902,A -85,B 0,C 180,E1 -19328.788,E2 -19328.788} C_VEL
LIN {X 0,Y 250.737,Z 497.249,A -85,B 0,C 180,E1 -19330.771,E2 -19330.771} C_VEL
LIN {X 0,Y 248.714,Z 505.363,A -85,B 0,C 180,E1 -19333.164,E2 -19333.164} C_VEL
LIN {X 0,Y 246.812,Z 512.469,A -85,B 0,C 180,E1 -19335.821,E2 -19335.821} C_VEL
LIN {X 0,Y 245.451,Z 517.84,A -85,B 0,C 180,E1 -19338.438,E2 -19338.438} C_VEL
LIN {X 0,Y 244.2,Z 521.73,A -85,B 0,C 180,E1 -19340.893,E2 -19340.893} C_VEL
LIN {X 0,Y 243.203,Z 524.607,A -85,B 0,C 180,E1 -19343.362,E2 -19343.362} C_VEL
LIN {X 0,Y 243.005,Z 525.944,A -85,B 0,C 180,E1 -19345.023,E2 -19345.023} C_VEL
LIN {X 0,Y 242.686,Z 526.919,A -85,B 0,C 180,E1 -19346.68,E2 -19346.68} C_VEL
LIN {X 0,Y 242.654,Z 527.496,A -85,B 0,C 180,E1 -19348.34,E2 -19348.34} C_VEL
LIN {X 0,Y 242.609,Z 527.72,A -85,B 0,C 180,E1 -19350,E2 -19350} C_VEL
LIN {X 0,Y 242.654,Z 527.532,A -85,B 0,C 180,E1 -19351.66,E2 -19351.66} C_VEL
LIN {X 0,Y 242.685,Z 526.977,A -85,B 0,C 180,E1 -19353.32,E2 -19353.32} C_VEL
LIN {X 0,Y 242.999,Z 526.026,A -85,B 0,C 180,E1 -19354.977,E2 -19354.977} C_VEL
LIN {X 0,Y 243.188,Z 524.727,A -85,B 0,C 180,E1 -19356.638,E2 -19356.638} C_VEL
LIN {X 0,Y 244.193,Z 521.893,A -85,B 0,C 180,E1 -19359.108,E2 -19359.108} C_VEL
LIN {X 0,Y 245.425,Z 518.061,A -85,B 0,C 180,E1 -19361.563,E2 -19361.563} C_VEL
LIN {X 0,Y 246.721,Z 512.977,A -85,B 0,C 180,E1 -19364.095,E2 -19364.095} C_VEL
LIN {X 0,Y 248.724,Z 505.73,A -85,B 0,C 180,E1 -19366.835,E2 -19366.835} C_VEL
LIN {X 0,Y 250.723,Z 497.698,A -85,B 0,C 180,E1 -19369.23,E2 -19369.23} C_VEL
LIN {X 0,Y 252.503,Z 489.47,A -85,B 0,C 180,E1 -19371.212,E2 -19371.212} C_VEL
LIN {X 0,Y 254.3,Z 480.425,A -85,B 0,C 180,E1 -19372.977,E2 -19372.977} C_VEL
LIN {X 0,Y 256.52,Z 468.872,A -85,B 0,C 180,E1 -19374.734,E2 -19374.734} C_VEL
LIN {X 0,Y 258.185,Z 456.928,A -85,B 0,C 180,E1 -19376.17,E2 -19376.17} C_VEL
LIN {X 0,Y 259.529,Z 444.316,A -85,B 0,C 180,E1 -19377.29,E2 -19377.29} C_VEL
LIN {X 0,Y 260.269,Z 432.226,A -85,B 0,C 180,E1 -19378.075,E2 -19378.075} C_VEL
LIN {X 0,Y 260.484,Z 420.949,A -85,B 0,C 180,E1 -19378.574,E2 -19378.574} C_VEL
LIN {X 0,Y 261.47,Z 379.087,A -85,B 0,C 180,E1 -19379.761,E2 -19379.761} C_VEL
LIN {X 0,Y 254.21,Z 363.897,A -85,B 0,C 180,E1 -19381.233,E2 -19381.233} C_VEL
LIN {X 0,Y 245.711,Z 348.522,A -85,B 0,C 180,E1 -19383.019,E2 -19383.019} C_VEL
LIN {X 0,Y 242.196,Z 342.359,A -85,B 0,C 180,E1 -19383.834,E2 -19383.834} C_VEL
LIN {X 0,Y 242.026,Z 341.417,A -85,B 0,C 180,E1 -19384.221,E2 -19384.221} C_VEL
LIN {X 0,Y 241.973,Z 341.323,A -85,B 0,C 180,E1 -19388.353,E2 -19388.353} C_VEL
LIN {X 0,Y 241.9,Z 341.318,A -85,B 0,C 180,E1 -19393.42,E2 -19393.42} C_VEL
LIN {X 0,Y 241.906,Z 341.341,A -85,B 0,C 180,E1 -19398.071,E2 -19398.071} C_VEL
LIN {X 0,Y 241.981,Z 341.305,A -85,B 0,C 180,E1 -19402.416,E2 -19402.416} C_VEL
LIN {X 0,Y 241.976,Z 341.336,A -85,B 0,C 180,E1 -19406.506,E2 -19406.506} C_VEL
LIN {X 0,Y 241.967,Z 341.278,A -85,B 0,C 180,E1 -19410.615,E2 -19410.615} C_VEL
LIN {X 0,Y 241.992,Z 341.329,A -85,B 0,C 180,E1 -19414.197,E2 -19414.197} C_VEL
LIN {X 0,Y 241.982,Z 341.326,A -85,B 0,C 180,E1 -19418.338,E2 -19418.338} C_VEL
LIN {X 0,Y 242.11,Z 341.323,A -85,B 0,C 180,E1 -19423.318,E2 -19423.318} C_VEL
LIN {X 0,Y 242.162,Z 341.319,A -85,B 0,C 180,E1 -19428.278,E2 -19428.278} C_VEL
LIN {X 0,Y 242.366,Z 341.274,A -85,B 0,C 180,E1 -19431.663,E2 -19431.663} C_VEL
LIN {X 0,Y 242.391,Z 341.276,A -85,B 0,C 180,E1 -19433.34,E2 -19433.34} C_VEL
LIN {X 0,Y 242.613,Z 341.243,A -85,B 0,C 180,E1 -19438.34,E2 -19438.34} C_VEL
LIN {X 0,Y 242.615,Z 341.259,A -85,B 0,C 180,E1 -19441.66,E2 -19441.66} C_VEL
LIN {X 0,Y 242.394,Z 341.27,A -85,B 0,C 180,E1 -19446.66,E2 -19446.66} C_VEL
LIN {X 0,Y 242.262,Z 341.307,A -85,B 0,C 180,E1 -19450.024,E2 -19450.024} C_VEL
LIN {X 0,Y 242.134,Z 341.322,A -85,B 0,C 180,E1 -19455.143,E2 -19455.143} C_VEL
LIN {X 0,Y 242.045,Z 341.312,A -85,B 0,C 180,E1 -19458.626,E2 -19458.626} C_VEL
LIN {X 0,Y 241.971,Z 341.321,A -85,B 0,C 180,E1 -19462.886,E2 -19462.886} C_VEL
LIN {X 0,Y 241.304,Z 341.427,A -85,B 0,C 180,E1 -19464.273,E2 -19464.273} C_VEL
LIN {X 0,Y 238.464,Z 341.767,A -85,B 0,C 180,E1 -19466.537,E2 -19466.537} C_VEL
LIN {X 0,Y 236.042,Z 342.058,A -85,B 0,C 180,E1 -19468.382,E2 -19468.382} C_VEL
LIN {X 0,Y 234.992,Z 342.193,A -85,B 0,C 180,E1 -19469.813,E2 -19469.813} C_VEL
LIN {X 0,Y 234.9,Z 342.211,A -85,B 0,C 180,E1 -19470.298,E2 -19470.298} C_VEL
LIN {X 0,Y 234.938,Z 342.208,A -85,B 0,C 180,E1 -19473.114,E2 -19473.114} C_VEL
LIN {X 0,Y 234.913,Z 342.222,A -85,B 0,C 180,E1 -19476.752,E2 -19476.752} C_VEL
LIN {X 0,Y 234.909,Z 342.208,A -85,B 0,C 180,E1 -19478.936,E2 -19478.936} C_VEL
LIN {X 0,Y 234.89,Z 342.375,A -85,B 0,C 180,E1 -19483.16,E2 -19483.16} C_VEL
LIN {X 0,Y 237.712,Z 352.227,A -85,B 0,C 180,E1 -19487.157,E2 -19487.157} C_VEL
LIN {X 0,Y 240.289,Z 362.049,A -85,B 0,C 180,E1 -19490.811,E2 -19490.811} C_VEL
LIN {X 0,Y 242.715,Z 373.102,A -85,B 0,C 180,E1 -19494.612,E2 -19494.612} C_VEL
LIN {X 0,Y 243.425,Z 376.626,A -85,B 0,C 180,E1 -19495.654,E2 -19495.654} C_VEL
LIN {X 0,Y 245.08,Z 381.419,A -85,B 0,C 180,E1 -19496.102,E2 -19496.102} C_VEL
LIN {X 0,Y 248.763,Z 410.099,A -85,B 0,C 180,E1 -19497.605,E2 -19497.605} C_VEL
LIN {X 0,Y 251.814,Z 441.46,A -85,B 0,C 180,E1 -19499.046,E2 -19499.046} C_VEL
LIN {X 0,Y 252.743,Z 455.97,A -85,B 0,C 180,E1 -19499.632,E2 -19499.632} C_VEL
LIN {X 0,Y 251.508,Z 489.046,A -85,B 0,C 180,E1 -19500.596,E2 -19500.596} C_VEL
LIN {X 0,Y 250.264,Z 502.398,A -85,B 0,C 180,E1 -19501.276,E2 -19501.276} C_VEL
LIN {X 0,Y 248.64,Z 514.639,A -85,B 0,C 180,E1 -19502.201,E2 -19502.201} C_VEL
LIN {X 0,Y 246.679,Z 525.81,A -85,B 0,C 180,E1 -19503.339,E2 -19503.339} C_VEL
LIN {X 0,Y 244.167,Z 537.456,A -85,B 0,C 180,E1 -19504.878,E2 -19504.878} C_VEL
LIN {X 0,Y 241.666,Z 547.977,A -85,B 0,C 180,E1 -19506.657,E2 -19506.657} C_VEL
LIN {X 0,Y 239.539,Z 556.617,A -85,B 0,C 180,E1 -19508.485,E2 -19508.485} C_VEL
LIN {X 0,Y 237.553,Z 564.626,A -85,B 0,C 180,E1 -19510.56,E2 -19510.56} C_VEL
LIN {X 0,Y 235.616,Z 572.486,A -85,B 0,C 180,E1 -19513.093,E2 -19513.093} C_VEL
LIN {X 0,Y 234.698,Z 577.946,A -85,B 0,C 180,E1 -19515.254,E2 -19515.254} C_VEL
LIN {X 0,Y 233.884,Z 583.262,A -85,B 0,C 180,E1 -19517.858,E2 -19517.858} C_VEL
LIN {X 0,Y 233.615,Z 587.448,A -85,B 0,C 180,E1 -19520.476,E2 -19520.476} C_VEL
LIN {X 0,Y 233.778,Z 590.593,A -85,B 0,C 180,E1 -19523.094,E2 -19523.094} C_VEL
LIN {X 0,Y 234.057,Z 592.119,A -85,B 0,C 180,E1 -19524.832,E2 -19524.832} C_VEL
LIN {X 0,Y 234.369,Z 593.223,A -85,B 0,C 180,E1 -19526.562,E2 -19526.562} C_VEL
LIN {X 0,Y 235.157,Z 594.203,A -85,B 0,C 180,E1 -19530,E2 -19530} C_VEL
LIN {X 0,Y 234.381,Z 593.209,A -85,B 0,C 180,E1 -19533.438,E2 -19533.438} C_VEL
LIN {X 0,Y 234.08,Z 592.101,A -85,B 0,C 180,E1 -19535.168,E2 -19535.168} C_VEL
LIN {X 0,Y 233.763,Z 590.253,A -85,B 0,C 180,E1 -19537.19,E2 -19537.19} C_VEL
LIN {X 0,Y 233.639,Z 586.093,A -85,B 0,C 180,E1 -19540.398,E2 -19540.398} C_VEL
LIN {X 0,Y 234.102,Z 581.527,A -85,B 0,C 180,E1 -19543.012,E2 -19543.012} C_VEL
LIN {X 0,Y 235.053,Z 575.773,A -85,B 0,C 180,E1 -19545.61,E2 -19545.61} C_VEL
LIN {X 0,Y 236.205,Z 570.018,A -85,B 0,C 180,E1 -19547.723,E2 -19547.723} C_VEL
LIN {X 0,Y 238.267,Z 561.448,A -85,B 0,C 180,E1 -19550.278,E2 -19550.278} C_VEL
LIN {X 0,Y 240.434,Z 552.804,A -85,B 0,C 180,E1 -19552.333,E2 -19552.333} C_VEL
LIN {X 0,Y 242.961,Z 542.168,A -85,B 0,C 180,E1 -19554.343,E2 -19554.343} C_VEL
LIN {X 0,Y 245.685,Z 530.254,A -85,B 0,C 180,E1 -19556.091,E2 -19556.091} C_VEL
LIN {X 0,Y 247.974,Z 518.263,A -85,B 0,C 180,E1 -19557.422,E2 -19557.422} C_VEL
LIN {X 0,Y 249.754,Z 505.786,A -85,B 0,C 180,E1 -19558.464,E2 -19558.464} C_VEL
LIN {X 0,Y 251.154,Z 492.752,A -85,B 0,C 180,E1 -19559.216,E2 -19559.216} C_VEL
LIN {X 0,Y 251.929,Z 477.819,A -85,B 0,C 180,E1 -19559.729,E2 -19559.729} C_VEL
LIN {X 0,Y 252.668,Z 454.985,A -85,B 0,C 180,E1 -19560.364,E2 -19560.364} C_VEL
LIN {X 0,Y 250.114,Z 423.463,A -85,B 0,C 180,E1 -19561.719,E2 -19561.719} C_VEL
LIN {X 0,Y 246.757,Z 394.185,A -85,B 0,C 180,E1 -19563.164,E2 -19563.164} C_VEL
LIN {X 0,Y 244.69,Z 380.023,A -85,B 0,C 180,E1 -19563.953,E2 -19563.953} C_VEL
LIN {X 0,Y 243.382,Z 376.29,A -85,B 0,C 180,E1 -19564.34,E2 -19564.34} C_VEL
LIN {X 0,Y 241.192,Z 366.07,A -85,B 0,C 180,E1 -19567.727,E2 -19567.727} C_VEL
LIN {X 0,Y 238.746,Z 355.957,A -85,B 0,C 180,E1 -19571.353,E2 -19571.353} C_VEL
LIN {X 0,Y 235.877,Z 345.833,A -85,B 0,C 180,E1 -19575.324,E2 -19575.324} C_VEL
LIN {X 0,Y 234.87,Z 342.331,A -85,B 0,C 180,E1 -19576.836,E2 -19576.836} C_VEL
LIN {X 0,Y 234.915,Z 342.158,A -85,B 0,C 180,E1 -19581.078,E2 -19581.078} C_VEL
LIN {X 0,Y 234.899,Z 342.17,A -85,B 0,C 180,E1 -19585.357,E2 -19585.357} C_VEL
LIN {X 0,Y 234.95,Z 342.215,A -85,B 0,C 180,E1 -19587.423,E2 -19587.423} C_VEL
LIN {X 0,Y 234.895,Z 342.196,A -85,B 0,C 180,E1 -19591.398,E2 -19591.398} C_VEL
LIN {X 0,Y 234.927,Z 342.223,A -85,B 0,C 180,E1 -19595.24,E2 -19595.24} C_VEL
LIN {X 0,Y 234.989,Z 342.172,A -85,B 0,C 180,E1 -19598.968,E2 -19598.968} C_VEL
LIN {X 0,Y 235.092,Z 342.199,A -85,B 0,C 180,E1 -19603.06,E2 -19603.06} C_VEL
LIN {X 0,Y 235.098,Z 342.181,A -85,B 0,C 180,E1 -19607.921,E2 -19607.921} C_VEL
LIN {X 0,Y 235.317,Z 342.169,A -85,B 0,C 180,E1 -19611.412,E2 -19611.412} C_VEL
LIN {X 0,Y 235.353,Z 342.148,A -85,B 0,C 180,E1 -19613.14,E2 -19613.14} C_VEL
LIN {X 0,Y 235.574,Z 342.137,A -85,B 0,C 180,E1 -19618.29,E2 -19618.29} C_VEL
LIN {X 0,Y 235.573,Z 342.119,A -85,B 0,C 180,E1 -19621.71,E2 -19621.71} C_VEL
LIN {X 0,Y 235.343,Z 342.15,A -85,B 0,C 180,E1 -19626.861,E2 -19626.861} C_VEL
LIN {X 0,Y 235.208,Z 342.183,A -85,B 0,C 180,E1 -19630.328,E2 -19630.328} C_VEL
LIN {X 0,Y 235.076,Z 342.184,A -85,B 0,C 180,E1 -19635.609,E2 -19635.609} C_VEL
LIN {X 0,Y 234.985,Z 342.206,A -85,B 0,C 180,E1 -19639.208,E2 -19639.208} C_VEL
LIN {X 0,Y 234.92,Z 342.218,A -85,B 0,C 180,E1 -19642.887,E2 -19642.887} C_VEL
LIN {X 0,Y 234.918,Z 342.192,A -85,B 0,C 180,E1 -19646.664,E2 -19646.664} C_VEL
LIN {X 0,Y 234.891,Z 342.162,A -85,B 0,C 180,E1 -19650.574,E2 -19650.574} C_VEL
LIN {X 0,Y 234.92,Z 342.223,A -85,B 0,C 180,E1 -19654.64,E2 -19654.64} C_VEL
LIN {X 0,Y 234.91,Z 342.174,A -85,B 0,C 180,E1 -19658.936,E2 -19658.936} C_VEL
LIN {X 0,Y 234.851,Z 342.232,A -85,B 0,C 180,E1 -19663.495,E2 -19663.495} C_VEL
LIN {X 0,Y 234.851,Z 342.195,A -85,B 0,C 180,E1 -19666.507,E2 -19666.507} C_VEL
LIN {X 0,Y 234.917,Z 342.209,A -85,B 0,C 180,E1 -19671.079,E2 -19671.079} C_VEL
LIN {X 0,Y 234.968,Z 342.38,A -85,B 0,C 180,E1 -19674.847,E2 -19674.847} C_VEL
LIN {X 0,Y 235.213,Z 343.398,A -85,B 0,C 180,E1 -19675.176,E2 -19675.176} C_VEL
LIN {X 0,Y 236.63,Z 346.011,A -85,B 0,C 180,E1 -19675.544,E2 -19675.544} C_VEL
LIN {X 0,Y 244.999,Z 360.32,A -85,B 0,C 180,E1 -19677.421,E2 -19677.421} C_VEL
LIN {X 0,Y 253.063,Z 376.209,A -85,B 0,C 180,E1 -19679.146,E2 -19679.146} C_VEL
LIN {X 0,Y 255.237,Z 381.089,A -85,B 0,C 180,E1 -19679.607,E2 -19679.607} C_VEL
LIN {X 0,Y 254.291,Z 421.25,A -85,B 0,C 180,E1 -19680.775,E2 -19680.775} C_VEL
LIN {X 0,Y 253.808,Z 434.842,A -85,B 0,C 180,E1 -19681.384,E2 -19681.384} C_VEL
LIN {X 0,Y 252.903,Z 447.46,A -85,B 0,C 180,E1 -19682.26,E2 -19682.26} C_VEL
LIN {X 0,Y 251.521,Z 459.689,A -85,B 0,C 180,E1 -19683.445,E2 -19683.445} C_VEL
LIN {X 0,Y 249.959,Z 469.948,A -85,B 0,C 180,E1 -19684.721,E2 -19684.721} C_VEL
LIN {X 0,Y 247.903,Z 480.692,A -85,B 0,C 180,E1 -19686.395,E2 -19686.395} C_VEL
LIN {X 0,Y 245.963,Z 489.884,A -85,B 0,C 180,E1 -19688.195,E2 -19688.195} C_VEL
LIN {X 0,Y 244.111,Z 498.23,A -85,B 0,C 180,E1 -19690.228,E2 -19690.228} C_VEL
LIN {X 0,Y 241.995,Z 506.343,A -85,B 0,C 180,E1 -19692.682,E2 -19692.682} C_VEL
LIN {X 0,Y 240.004,Z 513.449,A -85,B 0,C 180,E1 -19695.41,E2 -19695.41} C_VEL
LIN {X 0,Y 238.569,Z 518.819,A -85,B 0,C 180,E1 -19698.1,E2 -19698.1} C_VEL
LIN {X 0,Y 237.263,Z 522.708,A -85,B 0,C 180,E1 -19700.624,E2 -19700.624} C_VEL
LIN {X 0,Y 236.219,Z 525.586,A -85,B 0,C 180,E1 -19703.165,E2 -19703.165} C_VEL
LIN {X 0,Y 236.003,Z 526.923,A -85,B 0,C 180,E1 -19704.875,E2 -19704.875} C_VEL
LIN {X 0,Y 235.67,Z 527.897,A -85,B 0,C 180,E1 -19706.581,E2 -19706.581} C_VEL
LIN {X 0,Y 235.63,Z 528.474,A -85,B 0,C 180,E1 -19708.291,E2 -19708.291} C_VEL
LIN {X 0,Y 235.581,Z 528.698,A -85,B 0,C 180,E1 -19710,E2 -19710} C_VEL
LIN {X 0,Y 235.629,Z 528.509,A -85,B 0,C 180,E1 -19711.709,E2 -19711.709} C_VEL
LIN {X 0,Y 235.669,Z 527.955,A -85,B 0,C 180,E1 -19713.419,E2 -19713.419} C_VEL
LIN {X 0,Y 235.997,Z 527.004,A -85,B 0,C 180,E1 -19715.126,E2 -19715.126} C_VEL
LIN {X 0,Y 236.205,Z 525.705,A -85,B 0,C 180,E1 -19716.835,E2 -19716.835} C_VEL
LIN {X 0,Y 237.256,Z 522.87,A -85,B 0,C 180,E1 -19719.376,E2 -19719.376} C_VEL
LIN {X 0,Y 238.544,Z 519.038,A -85,B 0,C 180,E1 -19721.902,E2 -19721.902} C_VEL
LIN {X 0,Y 239.91,Z 513.953,A -85,B 0,C 180,E1 -19724.504,E2 -19724.504} C_VEL
LIN {X 0,Y 242.006,Z 506.706,A -85,B 0,C 180,E1 -19727.317,E2 -19727.317} C_VEL
LIN {X 0,Y 244.098,Z 498.673,A -85,B 0,C 180,E1 -19729.773,E2 -19729.773} C_VEL
LIN {X 0,Y 245.962,Z 490.445,A -85,B 0,C 180,E1 -19731.805,E2 -19731.805} C_VEL
LIN {X 0,Y 247.844,Z 481.399,A -85,B 0,C 180,E1 -19733.611,E2 -19733.611} C_VEL
LIN {X 0,Y 250.151,Z 469.844,A -85,B 0,C 180,E1 -19735.408,E2 -19735.408} C_VEL
LIN {X 0,Y 251.894,Z 457.9,A -85,B 0,C 180,E1 -19736.875,E2 -19736.875} C_VEL
LIN {X 0,Y 253.297,Z 445.286,A -85,B 0,C 180,E1 -19738.019,E2 -19738.019} C_VEL
LIN {X 0,Y 254.095,Z 432.941,A -85,B 0,C 180,E1 -19738.835,E2 -19738.835} C_VEL
LIN {X 0,Y 254.307,Z 421.66,A -85,B 0,C 180,E1 -19739.344,E2 -19739.344} C_VEL
LIN {X 0,Y 255.322,Z 381.168,A -85,B 0,C 180,E1 -19740.517,E2 -19740.517} C_VEL
LIN {X 0,Y 248.25,Z 366.412,A -85,B 0,C 180,E1 -19742.018,E2 -19742.018} C_VEL
LIN {X 0,Y 239.081,Z 349.956,A -85,B 0,C 180,E1 -19744.045,E2 -19744.045} C_VEL
LIN {X 0,Y 236.368,Z 345.661,A -85,B 0,C 180,E1 -19744.663,E2 -19744.663} C_VEL
LIN {X 0,Y 235.078,Z 342.927,A -85,B 0,C 180,E1 -19745.07,E2 -19745.07} C_VEL
LIN {X 0,Y 234.959,Z 342.282,A -85,B 0,C 180,E1 -19745.418,E2 -19745.418} C_VEL
LIN {X 0,Y 234.911,Z 342.208,A -85,B 0,C 180,E1 -19748.934,E2 -19748.934} C_VEL
LIN {X 0,Y 234.861,Z 342.197,A -85,B 0,C 180,E1 -19754.095,E2 -19754.095} C_VEL
LIN {X 0,Y 234.851,Z 342.201,A -85,B 0,C 180,E1 -19758.825,E2 -19758.825} C_VEL
LIN {X 0,Y 234.916,Z 342.174,A -85,B 0,C 180,E1 -19761.078,E2 -19761.078} C_VEL
LIN {X 0,Y 234.92,Z 342.223,A -85,B 0,C 180,E1 -19765.36,E2 -19765.36} C_VEL
LIN {X 0,Y 234.891,Z 342.163,A -85,B 0,C 180,E1 -19769.426,E2 -19769.426} C_VEL
LIN {X 0,Y 234.936,Z 342.198,A -85,B 0,C 180,E1 -19773.821,E2 -19773.821} C_VEL
LIN {X 0,Y 234.935,Z 342.201,A -85,B 0,C 180,E1 -19778.963,E2 -19778.963} C_VEL
LIN {X 0,Y 235.051,Z 342.202,A -85,B 0,C 180,E1 -19783.093,E2 -19783.093} C_VEL
LIN {X 0,Y 235.094,Z 342.197,A -85,B 0,C 180,E1 -19787.921,E2 -19787.921} C_VEL
LIN {X 0,Y 235.306,Z 342.154,A -85,B 0,C 180,E1 -19791.411,E2 -19791.411} C_VEL
LIN {X 0,Y 235.342,Z 342.151,A -85,B 0,C 180,E1 -19793.139,E2 -19793.139} C_VEL
LIN {X 0,Y 235.572,Z 342.119,A -85,B 0,C 180,E1 -19798.29,E2 -19798.29} C_VEL
LIN {X 0,Y 235.573,Z 342.137,A -85,B 0,C 180,E1 -19801.71,E2 -19801.71} C_VEL
LIN {X 0,Y 235.345,Z 342.148,A -85,B 0,C 180,E1 -19806.86,E2 -19806.86} C_VEL
LIN {X 0,Y 235.208,Z 342.183,A -85,B 0,C 180,E1 -19810.328,E2 -19810.328} C_VEL
LIN {X 0,Y 235.081,Z 342.201,A -85,B 0,C 180,E1 -19815.609,E2 -19815.609} C_VEL
LIN {X 0,Y 234.985,Z 342.181,A -85,B 0,C 180,E1 -19819.208,E2 -19819.208} C_VEL
LIN {X 0,Y 234.935,Z 342.201,A -85,B 0,C 180,E1 -19822.886,E2 -19822.886} C_VEL
LIN {X 0,Y 234.924,Z 342.205,A -85,B 0,C 180,E1 -19826.663,E2 -19826.663} C_VEL
LIN {X 0,Y 234.9,Z 342.211,A -85,B 0,C 180,E1 -19830.298,E2 -19830.298} C_VEL
LIN {X 0,Y 234.211,Z 342.314,A -85,B 0,C 180,E1 -19831.728,E2 -19831.728} C_VEL
LIN {X 0,Y 231.346,Z 342.674,A -85,B 0,C 180,E1 -19834.061,E2 -19834.061} C_VEL
LIN {X 0,Y 228.933,Z 342.965,A -85,B 0,C 180,E1 -19835.962,E2 -19835.962} C_VEL
LIN {X 0,Y 227.911,Z 343.095,A -85,B 0,C 180,E1 -19837.439,E2 -19837.439} C_VEL
LIN {X 0,Y 227.835,Z 343.096,A -85,B 0,C 180,E1 -19837.939,E2 -19837.939} C_VEL
LIN {X 0,Y 227.85,Z 343.284,A -85,B 0,C 180,E1 -19842.082,E2 -19842.082} C_VEL
LIN {X 0,Y 230.729,Z 353.295,A -85,B 0,C 180,E1 -19846.353,E2 -19846.353} C_VEL
LIN {X 0,Y 233.187,Z 362.549,A -85,B 0,C 180,E1 -19849.951,E2 -19849.951} C_VEL
LIN {X 0,Y 235.502,Z 372.901,A -85,B 0,C 180,E1 -19853.683,E2 -19853.683} C_VEL
LIN {X 0,Y 236.036,Z 375.312,A -85,B 0,C 180,E1 -19854.411,E2 -19854.411} C_VEL
LIN {X 0,Y 239.274,Z 383.379,A -85,B 0,C 180,E1 -19855.266,E2 -19855.266} C_VEL
LIN {X 0,Y 242.809,Z 411.843,A -85,B 0,C 180,E1 -19856.802,E2 -19856.802} C_VEL
LIN {X 0,Y 245.994,Z 446.415,A -85,B 0,C 180,E1 -19858.425,E2 -19858.425} C_VEL
LIN {X 0,Y 246.552,Z 457.383,A -85,B 0,C 180,E1 -19858.864,E2 -19858.864} C_VEL
LIN {X 0,Y 245.381,Z 487.418,A -85,B 0,C 180,E1 -19859.753,E2 -19859.753} C_VEL
LIN {X 0,Y 244.091,Z 501.01,A -85,B 0,C 180,E1 -19860.447,E2 -19860.447} C_VEL
LIN {X 0,Y 242.388,Z 513.658,A -85,B 0,C 180,E1 -19861.419,E2 -19861.419} C_VEL
LIN {X 0,Y 240.34,Z 524.824,A -85,B 0,C 180,E1 -19862.577,E2 -19862.577} C_VEL
LIN {X 0,Y 237.715,Z 536.465,A -85,B 0,C 180,E1 -19864.146,E2 -19864.146} C_VEL
LIN {X 0,Y 235.169,Z 546.992,A -85,B 0,C 180,E1 -19865.972,E2 -19865.972} C_VEL
LIN {X 0,Y 232.891,Z 555.624,A -85,B 0,C 180,E1 -19867.839,E2 -19867.839} C_VEL
LIN {X 0,Y 230.803,Z 563.631,A -85,B 0,C 180,E1 -19869.967,E2 -19869.967} C_VEL
LIN {X 0,Y 228.88,Z 570.912,A -85,B 0,C 180,E1 -19872.351,E2 -19872.351} C_VEL
LIN {X 0,Y 227.771,Z 576.95,A -85,B 0,C 180,E1 -19874.795,E2 -19874.795} C_VEL
LIN {X 0,Y 226.875,Z 582.265,A -85,B 0,C 180,E1 -19877.477,E2 -19877.477} C_VEL
LIN {X 0,Y 226.555,Z 586.452,A -85,B 0,C 180,E1 -19880.177,E2 -19880.177} C_VEL
LIN {X 0,Y 226.686,Z 589.6,A -85,B 0,C 180,E1 -19882.876,E2 -19882.876} C_VEL
LIN {X 0,Y 226.953,Z 591.127,A -85,B 0,C 180,E1 -19884.67,E2 -19884.67} C_VEL
LIN {X 0,Y 227.305,Z 592.239,A -85,B 0,C 180,E1 -19886.455,E2 -19886.455} C_VEL
LIN {X 0,Y 228.115,Z 593.223,A -85,B 0,C 180,E1 -19890,E2 -19890} C_VEL
LIN {X 0,Y 227.318,Z 592.224,A -85,B 0,C 180,E1 -19893.545,E2 -19893.545} C_VEL
LIN {X 0,Y 226.976,Z 591.108,A -85,B 0,C 180,E1 -19895.33,E2 -19895.33} C_VEL
LIN {X 0,Y 226.691,Z 589.475,A -85,B 0,C 180,E1 -19897.214,E2 -19897.214} C_VEL
LIN {X 0,Y 226.616,Z 585.098,A -85,B 0,C 180,E1 -19900.724,E2 -19900.724} C_VEL
LIN {X 0,Y 227.136,Z 580.53,A -85,B 0,C 180,E1 -19903.418,E2 -19903.418} C_VEL
LIN {X 0,Y 228.166,Z 574.776,A -85,B 0,C 180,E1 -19906.094,E2 -19906.094} C_VEL
LIN {X 0,Y 229.092,Z 570.187,A -85,B 0,C 180,E1 -19907.865,E2 -19907.865} C_VEL
LIN {X 0,Y 231.166,Z 561.968,A -85,B 0,C 180,E1 -19910.464,E2 -19910.464} C_VEL
LIN {X 0,Y 233.347,Z 553.638,A -85,B 0,C 180,E1 -19912.582,E2 -19912.582} C_VEL
LIN {X 0,Y 235.957,Z 543.527,A -85,B 0,C 180,E1 -19914.644,E2 -19914.644} C_VEL
LIN {X 0,Y 238.65,Z 532.134,A -85,B 0,C 180,E1 -19916.449,E2 -19916.449} C_VEL
LIN {X 0,Y 240.984,Z 521.005,A -85,B 0,C 180,E1 -19917.815,E2 -19917.815} C_VEL
LIN {X 0,Y 243.065,Z 508.666,A -85,B 0,C 180,E1 -19918.967,E2 -19918.967} C_VEL
LIN {X 0,Y 244.621,Z 495.525,A -85,B 0,C 180,E1 -19919.834,E2 -19919.834} C_VEL
LIN {X 0,Y 245.568,Z 481.71,A -85,B 0,C 180,E1 -19920.412,E2 -19920.412} C_VEL
LIN {X 0,Y 246.446,Z 454.942,A -85,B 0,C 180,E1 -19921.182,E2 -19921.182} C_VEL
LIN {X 0,Y 243.95,Z 423.677,A -85,B 0,C 180,E1 -19922.576,E2 -19922.576} C_VEL
LIN {X 0,Y 240.824,Z 395.675,A -85,B 0,C 180,E1 -19924.004,E2 -19924.004} C_VEL
LIN {X 0,Y 238.959,Z 382.654,A -85,B 0,C 180,E1 -19924.755,E2 -19924.755} C_VEL
LIN {X 0,Y 235.948,Z 375.077,A -85,B 0,C 180,E1 -19925.576,E2 -19925.576} C_VEL
LIN {X 0,Y 233.703,Z 364.79,A -85,B 0,C 180,E1 -19929.161,E2 -19929.161} C_VEL
LIN {X 0,Y 231.333,Z 355.499,A -85,B 0,C 180,E1 -19932.701,E2 -19932.701} C_VEL
LIN {X 0,Y 228.535,Z 345.554,A -85,B 0,C 180,E1 -19936.824,E2 -19936.824} C_VEL
LIN {X 0,Y 227.831,Z 343.164,A -85,B 0,C 180,E1 -19937.988,E2 -19937.988} C_VEL
LIN {X 0,Y 227.837,Z 343.027,A -85,B 0,C 180,E1 -19941.907,E2 -19941.907} C_VEL
LIN {X 0,Y 227.873,Z 343.068,A -85,B 0,C 180,E1 -19946.378,E2 -19946.378} C_VEL
LIN {X 0,Y 227.872,Z 343.075,A -85,B 0,C 180,E1 -19950.431,E2 -19950.431} C_VEL
LIN {X 0,Y 227.876,Z 343.098,A -85,B 0,C 180,E1 -19954.42,E2 -19954.42} C_VEL
LIN {X 0,Y 227.948,Z 343.052,A -85,B 0,C 180,E1 -19958.286,E2 -19958.286} C_VEL
LIN {X 0,Y 228.03,Z 343.078,A -85,B 0,C 180,E1 -19962.827,E2 -19962.827} C_VEL
LIN {X 0,Y 228.057,Z 343.056,A -85,B 0,C 180,E1 -19967.542,E2 -19967.542} C_VEL
LIN {X 0,Y 228.256,Z 343.052,A -85,B 0,C 180,E1 -19971.144,E2 -19971.144} C_VEL
LIN {X 0,Y 228.305,Z 343.027,A -85,B 0,C 180,E1 -19972.927,E2 -19972.927} C_VEL
LIN {X 0,Y 228.532,Z 343.015,A -85,B 0,C 180,E1 -19978.238,E2 -19978.238} C_VEL
LIN {X 0,Y 228.531,Z 342.996,A -85,B 0,C 180,E1 -19981.762,E2 -19981.762} C_VEL
LIN {X 0,Y 228.296,Z 343.025,A -85,B 0,C 180,E1 -19987.073,E2 -19987.073} C_VEL
LIN {X 0,Y 228.138,Z 343.064,A -85,B 0,C 180,E1 -19990.652,E2 -19990.652} C_VEL
LIN {X 0,Y 228.034,Z 343.056,A -85,B 0,C 180,E1 -19994.274,E2 -19994.274} C_VEL
LIN {X 0,Y 227.95,Z 343.09,A -85,B 0,C 180,E1 -19997.958,E2 -19997.958} C_VEL
LIN {X 0,Y 227.903,Z 343.084,A -85,B 0,C 180,E1 -20002.315,E2 -20002.315} C_VEL
LIN {X 0,Y 227.897,Z 343.067,A -85,B 0,C 180,E1 -20006.582,E2 -20006.582} C_VEL
LIN {X 0,Y 227.866,Z 343.034,A -85,B 0,C 180,E1 -20010.279,E2 -20010.279} C_VEL
LIN {X 0,Y 227.873,Z 343.094,A -85,B 0,C 180,E1 -20013.721,E2 -20013.721} C_VEL
LIN {X 0,Y 227.838,Z 343.059,A -85,B 0,C 180,E1 -20018.093,E2 -20018.093} C_VEL
LIN {X 0,Y 227.783,Z 343.11,A -85,B 0,C 180,E1 -20022.749,E2 -20022.749} C_VEL
LIN {X 0,Y 227.783,Z 343.076,A -85,B 0,C 180,E1 -20027.252,E2 -20027.252} C_VEL
LIN {X 0,Y 227.838,Z 343.081,A -85,B 0,C 180,E1 -20031.909,E2 -20031.909} C_VEL
LIN {X 0,Y 227.904,Z 343.319,A -85,B 0,C 180,E1 -20033.637,E2 -20033.637} C_VEL
LIN {X 0,Y 228.202,Z 344.471,A -85,B 0,C 180,E1 -20033.947,E2 -20033.947} C_VEL
LIN {X 0,Y 229.783,Z 347.082,A -85,B 0,C 180,E1 -20034.36,E2 -20034.36} C_VEL
LIN {X 0,Y 238.091,Z 361.149,A -85,B 0,C 180,E1 -20036.34,E2 -20036.34} C_VEL
LIN {X 0,Y 246.3,Z 376.961,A -85,B 0,C 180,E1 -20038.189,E2 -20038.189} C_VEL
LIN {X 0,Y 249.127,Z 383.047,A -85,B 0,C 180,E1 -20038.81,E2 -20038.81} C_VEL
LIN {X 0,Y 248.171,Z 424.057,A -85,B 0,C 180,E1 -20040.053,E2 -20040.053} C_VEL
LIN {X 0,Y 247.633,Z 436.678,A -85,B 0,C 180,E1 -20040.656,E2 -20040.656} C_VEL
LIN {X 0,Y 246.704,Z 448.446,A -85,B 0,C 180,E1 -20041.5,E2 -20041.5} C_VEL
LIN {X 0,Y 245.254,Z 460.673,A -85,B 0,C 180,E1 -20042.711,E2 -20042.711} C_VEL
LIN {X 0,Y 243.623,Z 470.931,A -85,B 0,C 180,E1 -20044.015,E2 -20044.015} C_VEL
LIN {X 0,Y 241.48,Z 481.674,A -85,B 0,C 180,E1 -20045.727,E2 -20045.727} C_VEL
LIN {X 0,Y 239.45,Z 490.865,A -85,B 0,C 180,E1 -20047.57,E2 -20047.57} C_VEL
LIN {X 0,Y 237.509,Z 499.21,A -85,B 0,C 180,E1 -20049.654,E2 -20049.654} C_VEL
LIN {X 0,Y 235.295,Z 507.323,A -85,B 0,C 180,E1 -20052.173,E2 -20052.173} C_VEL
LIN {X 0,Y 233.209,Z 514.429,A -85,B 0,C 180,E1 -20054.975,E2 -20054.975} C_VEL
LIN {X 0,Y 231.697,Z 519.798,A -85,B 0,C 180,E1 -20057.741,E2 -20057.741} C_VEL
LIN {X 0,Y 230.332,Z 523.687,A -85,B 0,C 180,E1 -20060.339,E2 -20060.339} C_VEL
LIN {X 0,Y 229.239,Z 526.566,A -85,B 0,C 180,E1 -20062.956,E2 -20062.956} C_VEL
LIN {X 0,Y 229.002,Z 527.901,A -85,B 0,C 180,E1 -20064.717,E2 -20064.717} C_VEL
LIN {X 0,Y 228.655,Z 528.875,A -85,B 0,C 180,E1 -20066.476,E2 -20066.476} C_VEL
LIN {X 0,Y 228.605,Z 529.452,A -85,B 0,C 180,E1 -20068.238,E2 -20068.238} C_VEL
LIN {X 0,Y 228.554,Z 529.676,A -85,B 0,C 180,E1 -20070,E2 -20070} C_VEL
LIN {X 0,Y 228.605,Z 529.487,A -85,B 0,C 180,E1 -20071.762,E2 -20071.762} C_VEL
LIN {X 0,Y 228.654,Z 528.932,A -85,B 0,C 180,E1 -20073.524,E2 -20073.524} C_VEL
LIN {X 0,Y 228.996,Z 527.981,A -85,B 0,C 180,E1 -20075.283,E2 -20075.283} C_VEL
LIN {X 0,Y 229.224,Z 526.683,A -85,B 0,C 180,E1 -20077.044,E2 -20077.044} C_VEL
LIN {X 0,Y 230.325,Z 523.847,A -85,B 0,C 180,E1 -20079.661,E2 -20079.661} C_VEL
LIN {X 0,Y 231.672,Z 520.015,A -85,B 0,C 180,E1 -20082.26,E2 -20082.26} C_VEL
LIN {X 0,Y 233.113,Z 514.93,A -85,B 0,C 180,E1 -20084.937,E2 -20084.937} C_VEL
LIN {X 0,Y 235.306,Z 507.682,A -85,B 0,C 180,E1 -20087.827,E2 -20087.827} C_VEL
LIN {X 0,Y 237.495,Z 499.649,A -85,B 0,C 180,E1 -20090.347,E2 -20090.347} C_VEL
LIN {X 0,Y 239.449,Z 491.42,A -85,B 0,C 180,E1 -20092.43,E2 -20092.43} C_VEL
LIN {X 0,Y 241.406,Z 482.375,A -85,B 0,C 180,E1 -20094.281,E2 -20094.281} C_VEL
LIN {X 0,Y 243.828,Z 470.816,A -85,B 0,C 180,E1 -20096.116,E2 -20096.116} C_VEL
LIN {X 0,Y 245.647,Z 458.872,A -85,B 0,C 180,E1 -20097.616,E2 -20097.616} C_VEL
LIN {X 0,Y 247.108,Z 446.256,A -85,B 0,C 180,E1 -20098.786,E2 -20098.786} C_VEL
LIN {X 0,Y 247.916,Z 434.306,A -85,B 0,C 180,E1 -20099.599,E2 -20099.599} C_VEL
LIN {X 0,Y 248.202,Z 422.453,A -85,B 0,C 180,E1 -20100.146,E2 -20100.146} C_VEL
LIN {X 0,Y 249.228,Z 383.148,A -85,B 0,C 180,E1 -20101.312,E2 -20101.312} C_VEL
LIN {X 0,Y 241.195,Z 366.77,A -85,B 0,C 180,E1 -20103.1,E2 -20103.1} C_VEL
LIN {X 0,Y 232.076,Z 350.816,A -85,B 0,C 180,E1 -20105.232,E2 -20105.232} C_VEL
LIN {X 0,Y 229.385,Z 346.627,A -85,B 0,C 180,E1 -20105.886,E2 -20105.886} C_VEL
LIN {X 0,Y 228.02,Z 343.878,A -85,B 0,C 180,E1 -20106.321,E2 -20106.321} C_VEL
LIN {X 0,Y 227.888,Z 343.168,A -85,B 0,C 180,E1 -20106.694,E2 -20106.694} C_VEL
LIN {X 0,Y 227.794,Z 343.109,A -85,B 0,C 180,E1 -20110.383,E2 -20110.383} C_VEL
LIN {X 0,Y 227.808,Z 343.088,A -85,B 0,C 180,E1 -20115.198,E2 -20115.198} C_VEL
LIN {X 0,Y 227.798,Z 343.066,A -85,B 0,C 180,E1 -20119.617,E2 -20119.617} C_VEL
LIN {X 0,Y 227.863,Z 343.093,A -85,B 0,C 180,E1 -20124.125,E2 -20124.125} C_VEL
LIN {X 0,Y 227.85,Z 343.053,A -85,B 0,C 180,E1 -20128.374,E2 -20128.374} C_VEL
LIN {X 0,Y 227.837,Z 343.052,A -85,B 0,C 180,E1 -20132.438,E2 -20132.438} C_VEL
LIN {X 0,Y 227.861,Z 343.102,A -85,B 0,C 180,E1 -20136.361,E2 -20136.361} C_VEL
LIN {X 0,Y 227.891,Z 343.083,A -85,B 0,C 180,E1 -20140.17,E2 -20140.17} C_VEL
LIN {X 0,Y 228.014,Z 343.069,A -85,B 0,C 180,E1 -20143.894,E2 -20143.894} C_VEL
LIN {X 0,Y 228.138,Z 343.065,A -85,B 0,C 180,E1 -20149.348,E2 -20149.348} C_VEL
LIN {X 0,Y 228.295,Z 343.027,A -85,B 0,C 180,E1 -20152.927,E2 -20152.927} C_VEL
LIN {X 0,Y 228.531,Z 342.997,A -85,B 0,C 180,E1 -20158.238,E2 -20158.238} C_VEL
LIN {X 0,Y 228.531,Z 343.014,A -85,B 0,C 180,E1 -20161.762,E2 -20161.762} C_VEL
LIN {X 0,Y 228.297,Z 343.027,A -85,B 0,C 180,E1 -20167.073,E2 -20167.073} C_VEL
LIN {X 0,Y 228.138,Z 343.061,A -85,B 0,C 180,E1 -20170.651,E2 -20170.651} C_VEL
LIN {X 0,Y 228.036,Z 343.066,A -85,B 0,C 180,E1 -20174.274,E2 -20174.274} C_VEL
LIN {X 0,Y 227.965,Z 343.074,A -85,B 0,C 180,E1 -20177.956,E2 -20177.956} C_VEL
LIN {X 0,Y 227.912,Z 343.065,A -85,B 0,C 180,E1 -20182.32,E2 -20182.32} C_VEL
LIN {X 0,Y 227.902,Z 343.08,A -85,B 0,C 180,E1 -20186.584,E2 -20186.584} C_VEL
LIN {X 0,Y 227.87,Z 343.086,A -85,B 0,C 180,E1 -20190.281,E2 -20190.281} C_VEL
LIN {X 0,Y 227.873,Z 343.081,A -85,B 0,C 180,E1 -20193.721,E2 -20193.721} C_VEL
LIN {X 0,Y 227.835,Z 343.096,A -85,B 0,C 180,E1 -20197.939,E2 -20197.939} C_VEL
LIN {X 0,Y 227.194,Z 343.317,A -85,B 0,C 180,E1 -20198.942,E2 -20198.942} C_VEL
LIN {X 0,Y 224.562,Z 344.537,A -85,B 0,C 180,E1 -20200.514,E2 -20200.514} C_VEL
LIN {X 0,Y 222.562,Z 346.24,A -85,B 0,C 180,E1 -20201.743,E2 -20201.743} C_VEL
LIN {X 0,Y 221.995,Z 348.1,A -85,B 0,C 180,E1 -20202.745,E2 -20202.745} C_VEL
LIN {X 0,Y 222.095,Z 348.583,A -85,B 0,C 180,E1 -20202.971,E2 -20202.971} C_VEL
LIN {X 0,Y 224.374,Z 356.63,A -85,B 0,C 180,E1 -20206.442,E2 -20206.442} C_VEL
LIN {X 0,Y 226.802,Z 366.088,A -85,B 0,C 180,E1 -20210.213,E2 -20210.213} C_VEL
LIN {X 0,Y 228.531,Z 373.852,A -85,B 0,C 180,E1 -20213.029,E2 -20213.029} C_VEL
LIN {X 0,Y 233.142,Z 384.956,A -85,B 0,C 180,E1 -20214.31,E2 -20214.31} C_VEL
LIN {X 0,Y 233.813,Z 387.791,A -85,B 0,C 180,E1 -20214.527,E2 -20214.527} C_VEL
LIN {X 0,Y 236.811,Z 412.721,A -85,B 0,C 180,E1 -20215.913,E2 -20215.913} C_VEL
LIN {X 0,Y 239.814,Z 446.224,A -85,B 0,C 180,E1 -20217.54,E2 -20217.54} C_VEL
LIN {X 0,Y 240.45,Z 457.494,A -85,B 0,C 180,E1 -20218.019,E2 -20218.019} C_VEL
LIN {X 0,Y 239.224,Z 486.671,A -85,B 0,C 180,E1 -20218.902,E2 -20218.902} C_VEL
LIN {X 0,Y 237.929,Z 500.18,A -85,B 0,C 180,E1 -20219.614,E2 -20219.614} C_VEL
LIN {X 0,Y 236.158,Z 512.673,A -85,B 0,C 180,E1 -20220.592,E2 -20220.592} C_VEL
LIN {X 0,Y 234.036,Z 523.837,A -85,B 0,C 180,E1 -20221.774,E2 -20221.774} C_VEL
LIN {X 0,Y 231.319,Z 535.477,A -85,B 0,C 180,E1 -20223.376,E2 -20223.376} C_VEL
LIN {X 0,Y 228.614,Z 545.994,A -85,B 0,C 180,E1 -20225.238,E2 -20225.238} C_VEL
LIN {X 0,Y 226.287,Z 554.632,A -85,B 0,C 180,E1 -20227.156,E2 -20227.156} C_VEL
LIN {X 0,Y 224.091,Z 562.637,A -85,B 0,C 180,E1 -20229.34,E2 -20229.34} C_VEL
LIN {X 0,Y 222.348,Z 569.318,A -85,B 0,C 180,E1 -20231.574,E2 -20231.574} C_VEL
LIN {X 0,Y 220.842,Z 575.951,A -85,B 0,C 180,E1 -20234.306,E2 -20234.306} C_VEL
LIN {X 0,Y 219.884,Z 581.269,A -85,B 0,C 180,E1 -20237.072,E2 -20237.072} C_VEL
LIN {X 0,Y 219.497,Z 585.456,A -85,B 0,C 180,E1 -20239.857,E2 -20239.857} C_VEL
LIN {X 0,Y 219.624,Z 588.703,A -85,B 0,C 180,E1 -20242.751,E2 -20242.751} C_VEL
LIN {X 0,Y 220.238,Z 591.254,A -85,B 0,C 180,E1 -20246.341,E2 -20246.341} C_VEL
LIN {X 0,Y 221.072,Z 592.243,A -85,B 0,C 180,E1 -20250,E2 -20250} C_VEL
LIN {X 0,Y 220.251,Z 591.239,A -85,B 0,C 180,E1 -20253.659,E2 -20253.659} C_VEL
LIN {X 0,Y 219.628,Z 588.665,A -85,B 0,C 180,E1 -20257.258,E2 -20257.258} C_VEL
LIN {X 0,Y 219.499,Z 585.406,A -85,B 0,C 180,E1 -20260.143,E2 -20260.143} C_VEL
LIN {X 0,Y 219.881,Z 581.198,A -85,B 0,C 180,E1 -20262.929,E2 -20262.929} C_VEL
LIN {X 0,Y 221.039,Z 574.82,A -85,B 0,C 180,E1 -20266.153,E2 -20266.153} C_VEL
LIN {X 0,Y 222.329,Z 569.195,A -85,B 0,C 180,E1 -20268.427,E2 -20268.427} C_VEL
LIN {X 0,Y 224.494,Z 560.973,A -85,B 0,C 180,E1 -20271.101,E2 -20271.101} C_VEL
LIN {X 0,Y 226.786,Z 552.644,A -85,B 0,C 180,E1 -20273.273,E2 -20273.273} C_VEL
LIN {X 0,Y 229.447,Z 542.524,A -85,B 0,C 180,E1 -20275.392,E2 -20275.392} C_VEL
LIN {X 0,Y 232.318,Z 531.142,A -85,B 0,C 180,E1 -20277.229,E2 -20277.229} C_VEL
LIN {X 0,Y 234.73,Z 520.012,A -85,B 0,C 180,E1 -20278.623,E2 -20278.623} C_VEL
LIN {X 0,Y 236.836,Z 507.664,A -85,B 0,C 180,E1 -20279.804,E2 -20279.804} C_VEL
LIN {X 0,Y 238.485,Z 494.404,A -85,B 0,C 180,E1 -20280.691,E2 -20280.691} C_VEL
LIN {X 0,Y 239.452,Z 481.069,A -85,B 0,C 180,E1 -20281.26,E2 -20281.26} C_VEL
LIN {X 0,Y 240.335,Z 455.871,A -85,B 0,C 180,E1 -20282.002,E2 -20282.002} C_VEL
LIN {X 0,Y 238.003,Z 425.487,A -85,B 0,C 180,E1 -20283.397,E2 -20283.397} C_VEL
LIN {X 0,Y 235.165,Z 399.273,A -85,B 0,C 180,E1 -20284.775,E2 -20284.775} C_VEL
LIN {X 0,Y 233.234,Z 385.125,A -85,B 0,C 180,E1 -20285.61,E2 -20285.61} C_VEL
LIN {X 0,Y 228.546,Z 373.814,A -85,B 0,C 180,E1 -20286.915,E2 -20286.915} C_VEL
LIN {X 0,Y 226.189,Z 363.485,A -85,B 0,C 180,E1 -20290.729,E2 -20290.729} C_VEL
LIN {X 0,Y 223.438,Z 353.162,A -85,B 0,C 180,E1 -20294.951,E2 -20294.951} C_VEL
LIN {X 0,Y 220.768,Z 344.036,A -85,B 0,C 180,E1 -20299.137,E2 -20299.137} C_VEL
LIN {X 0,Y 220.822,Z 343.895,A -85,B 0,C 180,E1 -20302.792,E2 -20302.792} C_VEL
LIN {X 0,Y 220.808,Z 343.97,A -85,B 0,C 180,E1 -20307.242,E2 -20307.242} C_VEL
LIN {X 0,Y 220.796,Z 343.951,A -85,B 0,C 180,E1 -20311.481,E2 -20311.481} C_VEL
LIN {X 0,Y 220.829,Z 343.977,A -85,B 0,C 180,E1 -20315.561,E2 -20315.561} C_VEL
LIN {X 0,Y 220.879,Z 343.928,A -85,B 0,C 180,E1 -20319.513,E2 -20319.513} C_VEL
LIN {X 0,Y 221.01,Z 343.954,A -85,B 0,C 180,E1 -20323.37,E2 -20323.37} C_VEL
LIN {X 0,Y 221.06,Z 343.942,A -85,B 0,C 180,E1 -20329.003,E2 -20329.003} C_VEL
LIN {X 0,Y 221.242,Z 343.908,A -85,B 0,C 180,E1 -20332.7,E2 -20332.7} C_VEL
LIN {X 0,Y 221.465,Z 343.895,A -85,B 0,C 180,E1 -20338.182,E2 -20338.182} C_VEL
LIN {X 0,Y 221.465,Z 343.877,A -85,B 0,C 180,E1 -20341.819,E2 -20341.819} C_VEL
LIN {X 0,Y 221.234,Z 343.903,A -85,B 0,C 180,E1 -20347.3,E2 -20347.3} C_VEL
LIN {X 0,Y 221.059,Z 343.947,A -85,B 0,C 180,E1 -20350.997,E2 -20350.997} C_VEL
LIN {X 0,Y 220.976,Z 343.952,A -85,B 0,C 180,E1 -20356.633,E2 -20356.633} C_VEL
LIN {X 0,Y 220.866,Z 343.953,A -85,B 0,C 180,E1 -20360.489,E2 -20360.489} C_VEL
LIN {X 0,Y 220.801,Z 343.981,A -85,B 0,C 180,E1 -20364.443,E2 -20364.443} C_VEL
LIN {X 0,Y 220.791,Z 343.916,A -85,B 0,C 180,E1 -20368.52,E2 -20368.52} C_VEL
LIN {X 0,Y 220.808,Z 343.952,A -85,B 0,C 180,E1 -20372.758,E2 -20372.758} C_VEL
LIN {X 0,Y 220.799,Z 343.945,A -85,B 0,C 180,E1 -20377.276,E2 -20377.276} C_VEL
LIN {X 0,Y 220.746,Z 343.968,A -85,B 0,C 180,E1 -20381.959,E2 -20381.959} C_VEL
LIN {X 0,Y 220.751,Z 343.957,A -85,B 0,C 180,E1 -20385.541,E2 -20385.541} C_VEL
LIN {X 0,Y 220.78,Z 343.978,A -85,B 0,C 180,E1 -20390.458,E2 -20390.458} C_VEL
LIN {X 0,Y 220.839,Z 344.223,A -85,B 0,C 180,E1 -20392.284,E2 -20392.284} C_VEL
LIN {X 0,Y 221.167,Z 345.48,A -85,B 0,C 180,E1 -20392.601,E2 -20392.601} C_VEL
LIN {X 0,Y 222.846,Z 348.123,A -85,B 0,C 180,E1 -20393.063,E2 -20393.063} C_VEL
LIN {X 0,Y 230.333,Z 360.444,A -85,B 0,C 180,E1 -20394.968,E2 -20394.968} C_VEL
LIN {X 0,Y 237.567,Z 373.706,A -85,B 0,C 180,E1 -20396.704,E2 -20396.704} C_VEL
LIN {X 0,Y 243.059,Z 385.154,A -85,B 0,C 180,E1 -20397.978,E2 -20397.978} C_VEL
LIN {X 0,Y 242.058,Z 426.833,A -85,B 0,C 180,E1 -20399.288,E2 -20399.288} C_VEL
LIN {X 0,Y 241.46,Z 438.957,A -85,B 0,C 180,E1 -20399.918,E2 -20399.918} C_VEL
LIN {X 0,Y 240.318,Z 451.69,A -85,B 0,C 180,E1 -20400.911,E2 -20400.911} C_VEL
LIN {X 0,Y 238.794,Z 463.385,A -85,B 0,C 180,E1 -20402.145,E2 -20402.145} C_VEL
LIN {X 0,Y 236.861,Z 474.038,A -85,B 0,C 180,E1 -20403.573,E2 -20403.573} C_VEL
LIN {X 0,Y 234.54,Z 484.868,A -85,B 0,C 180,E1 -20405.433,E2 -20405.433} C_VEL
LIN {X 0,Y 232.529,Z 493.628,A -85,B 0,C 180,E1 -20407.334,E2 -20407.334} C_VEL
LIN {X 0,Y 230.522,Z 501.646,A -85,B 0,C 180,E1 -20409.476,E2 -20409.476} C_VEL
LIN {X 0,Y 228.282,Z 509.503,A -85,B 0,C 180,E1 -20412.07,E2 -20412.07} C_VEL
LIN {X 0,Y 226.429,Z 515.408,A -85,B 0,C 180,E1 -20414.514,E2 -20414.514} C_VEL
LIN {X 0,Y 224.834,Z 520.778,A -85,B 0,C 180,E1 -20417.361,E2 -20417.361} C_VEL
LIN {X 0,Y 223.407,Z 524.666,A -85,B 0,C 180,E1 -20420.037,E2 -20420.037} C_VEL
LIN {X 0,Y 222.262,Z 527.545,A -85,B 0,C 180,E1 -20422.734,E2 -20422.734} C_VEL
LIN {X 0,Y 222.003,Z 528.88,A -85,B 0,C 180,E1 -20424.55,E2 -20424.55} C_VEL
LIN {X 0,Y 221.64,Z 529.854,A -85,B 0,C 180,E1 -20426.364,E2 -20426.364} C_VEL
LIN {X 0,Y 221.58,Z 530.43,A -85,B 0,C 180,E1 -20428.182,E2 -20428.182} C_VEL
LIN {X 0,Y 221.526,Z 530.654,A -85,B 0,C 180,E1 -20430,E2 -20430} C_VEL
LIN {X 0,Y 221.58,Z 530.465,A -85,B 0,C 180,E1 -20431.818,E2 -20431.818} C_VEL
LIN {X 0,Y 221.639,Z 529.91,A -85,B 0,C 180,E1 -20433.636,E2 -20433.636} C_VEL
LIN {X 0,Y 221.996,Z 528.959,A -85,B 0,C 180,E1 -20435.45,E2 -20435.45} C_VEL
LIN {X 0,Y 222.247,Z 527.661,A -85,B 0,C 180,E1 -20437.267,E2 -20437.267} C_VEL
LIN {X 0,Y 223.4,Z 524.824,A -85,B 0,C 180,E1 -20439.964,E2 -20439.964} C_VEL
LIN {X 0,Y 224.809,Z 520.992,A -85,B 0,C 180,E1 -20442.64,E2 -20442.64} C_VEL
LIN {X 0,Y 226.33,Z 515.906,A -85,B 0,C 180,E1 -20445.395,E2 -20445.395} C_VEL
LIN {X 0,Y 228.625,Z 508.658,A -85,B 0,C 180,E1 -20448.366,E2 -20448.366} C_VEL
LIN {X 0,Y 230.918,Z 500.625,A -85,B 0,C 180,E1 -20450.953,E2 -20450.953} C_VEL
LIN {X 0,Y 232.966,Z 492.395,A -85,B 0,C 180,E1 -20453.09,E2 -20453.09} C_VEL
LIN {X 0,Y 234.996,Z 483.352,A -85,B 0,C 180,E1 -20454.988,E2 -20454.988} C_VEL
LIN {X 0,Y 237.534,Z 471.792,A -85,B 0,C 180,E1 -20456.862,E2 -20456.862} C_VEL
LIN {X 0,Y 239.441,Z 459.844,A -85,B 0,C 180,E1 -20458.396,E2 -20458.396} C_VEL
LIN {X 0,Y 240.966,Z 447.227,A -85,B 0,C 180,E1 -20459.591,E2 -20459.591} C_VEL
LIN {X 0,Y 241.819,Z 435.088,A -85,B 0,C 180,E1 -20460.436,E2 -20460.436} C_VEL
LIN {X 0,Y 242.175,Z 421.958,A -85,B 0,C 180,E1 -20461.033,E2 -20461.033} C_VEL
LIN {X 0,Y 243.175,Z 385.258,A -85,B 0,C 180,E1 -20462.144,E2 -20462.144} C_VEL
LIN {X 0,Y 235.879,Z 370.382,A -85,B 0,C 180,E1 -20463.846,E2 -20463.846} C_VEL
LIN {X 0,Y 227.434,Z 355.469,A -85,B 0,C 180,E1 -20465.913,E2 -20465.913} C_VEL
LIN {X 0,Y 222.794,Z 348.092,A -85,B 0,C 180,E1 -20467.108,E2 -20467.108} C_VEL
LIN {X 0,Y 221.191,Z 345.573,A -85,B 0,C 180,E1 -20467.549,E2 -20467.549} C_VEL
LIN {X 0,Y 220.837,Z 344.29,A -85,B 0,C 180,E1 -20467.88,E2 -20467.88} C_VEL
LIN {X 0,Y 220.785,Z 343.984,A -85,B 0,C 180,E1 -20468.369,E2 -20468.369} C_VEL
LIN {X 0,Y 220.74,Z 343.952,A -85,B 0,C 180,E1 -20472.922,E2 -20472.922} C_VEL
LIN {X 0,Y 220.742,Z 343.99,A -85,B 0,C 180,E1 -20477.076,E2 -20477.076} C_VEL
LIN {X 0,Y 220.779,Z 343.934,A -85,B 0,C 180,E1 -20480.457,E2 -20480.457} C_VEL
LIN {X 0,Y 220.823,Z 343.942,A -85,B 0,C 180,E1 -20482.792,E2 -20482.792} C_VEL
LIN {X 0,Y 220.808,Z 343.953,A -85,B 0,C 180,E1 -20487.242,E2 -20487.242} C_VEL
LIN {X 0,Y 220.792,Z 343.916,A -85,B 0,C 180,E1 -20491.48,E2 -20491.48} C_VEL
LIN {X 0,Y 220.799,Z 343.981,A -85,B 0,C 180,E1 -20495.557,E2 -20495.557} C_VEL
LIN {X 0,Y 220.847,Z 343.956,A -85,B 0,C 180,E1 -20499.509,E2 -20499.509} C_VEL
LIN {X 0,Y 220.972,Z 343.953,A -85,B 0,C 180,E1 -20503.367,E2 -20503.367} C_VEL
LIN {X 0,Y 221.058,Z 343.948,A -85,B 0,C 180,E1 -20509.003,E2 -20509.003} C_VEL
LIN {X 0,Y 221.233,Z 343.905,A -85,B 0,C 180,E1 -20512.7,E2 -20512.7} C_VEL
LIN {X 0,Y 221.464,Z 343.877,A -85,B 0,C 180,E1 -20518.181,E2 -20518.181} C_VEL
LIN {X 0,Y 221.465,Z 343.894,A -85,B 0,C 180,E1 -20521.818,E2 -20521.818} C_VEL
LIN {X 0,Y 221.235,Z 343.908,A -85,B 0,C 180,E1 -20527.3,E2 -20527.3} C_VEL
LIN {X 0,Y 221.059,Z 343.94,A -85,B 0,C 180,E1 -20530.997,E2 -20530.997} C_VEL
LIN {X 0,Y 220.987,Z 343.957,A -85,B 0,C 180,E1 -20536.632,E2 -20536.632} C_VEL
LIN {X 0,Y 220.868,Z 343.929,A -85,B 0,C 180,E1 -20540.488,E2 -20540.488} C_VEL
LIN {X 0,Y 220.829,Z 343.978,A -85,B 0,C 180,E1 -20544.439,E2 -20544.439} C_VEL
LIN {X 0,Y 220.796,Z 343.951,A -85,B 0,C 180,E1 -20548.519,E2 -20548.519} C_VEL
LIN {X 0,Y 220.809,Z 343.971,A -85,B 0,C 180,E1 -20552.757,E2 -20552.757} C_VEL
LIN {X 0,Y 220.8,Z 343.983,A -85,B 0,C 180,E1 -20557.276,E2 -20557.276} C_VEL
LIN {X 0,Y 220.789,Z 344.169,A -85,B 0,C 180,E1 -20560.919,E2 -20560.919} C_VEL
LIN {X 0,Y 222.095,Z 348.583,A -85,B 0,C 180,E1 -20562.971,E2 -20562.971} C_VEL
LIN {X 0,Y 222.386,Z 351.763,A -85,B 0,C 180,E1 -20564.25,E2 -20564.25} C_VEL
LIN {X 0,Y 221.157,Z 357.716,A -85,B 0,C 180,E1 -20566.271,E2 -20566.271} C_VEL
LIN {X 0,Y 219.952,Z 362.652,A -85,B 0,C 180,E1 -20567.889,E2 -20567.889} C_VEL
LIN {X 0,Y 219.727,Z 366.178,A -85,B 0,C 180,E1 -20569.147,E2 -20569.147} C_VEL
LIN {X 0,Y 219.888,Z 367.288,A -85,B 0,C 180,E1 -20569.576,E2 -20569.576} C_VEL
LIN {X 0,Y 221.148,Z 372.661,A -85,B 0,C 180,E1 -20571.588,E2 -20571.588} C_VEL
LIN {X 0,Y 227.537,Z 387.551,A -85,B 0,C 180,E1 -20573.424,E2 -20573.424} C_VEL
LIN {X 0,Y 228.132,Z 390.38,A -85,B 0,C 180,E1 -20573.638,E2 -20573.638} C_VEL
LIN {X 0,Y 230.935,Z 414.328,A -85,B 0,C 180,E1 -20575.016,E2 -20575.016} C_VEL
LIN {X 0,Y 233.796,Z 447.192,A -85,B 0,C 180,E1 -20576.667,E2 -20576.667} C_VEL
LIN {X 0,Y 234.31,Z 459.096,A -85,B 0,C 180,E1 -20577.168,E2 -20577.168} C_VEL
LIN {X 0,Y 233.122,Z 485.943,A -85,B 0,C 180,E1 -20578.007,E2 -20578.007} C_VEL
LIN {X 0,Y 231.734,Z 499.838,A -85,B 0,C 180,E1 -20578.765,E2 -20578.765} C_VEL
LIN {X 0,Y 229.807,Z 512.706,A -85,B 0,C 180,E1 -20579.822,E2 -20579.822} C_VEL
LIN {X 0,Y 227.433,Z 524.444,A -85,B 0,C 180,E1 -20581.13,E2 -20581.13} C_VEL
LIN {X 0,Y 224.645,Z 535.793,A -85,B 0,C 180,E1 -20582.772,E2 -20582.772} C_VEL
LIN {X 0,Y 221.871,Z 546.059,A -85,B 0,C 180,E1 -20584.683,E2 -20584.683} C_VEL
LIN {X 0,Y 219.228,Z 555.343,A -85,B 0,C 180,E1 -20586.877,E2 -20586.877} C_VEL
LIN {X 0,Y 216.617,Z 564.583,A -85,B 0,C 180,E1 -20589.637,E2 -20589.637} C_VEL
LIN {X 0,Y 214.631,Z 571.553,A -85,B 0,C 180,E1 -20592.261,E2 -20592.261} C_VEL
LIN {X 0,Y 213.549,Z 576.847,A -85,B 0,C 180,E1 -20594.735,E2 -20594.735} C_VEL
LIN {X 0,Y 212.685,Z 581.776,A -85,B 0,C 180,E1 -20597.597,E2 -20597.597} C_VEL
LIN {X 0,Y 212.42,Z 585.606,A -85,B 0,C 180,E1 -20600.478,E2 -20600.478} C_VEL
LIN {X 0,Y 212.572,Z 587.858,A -85,B 0,C 180,E1 -20602.682,E2 -20602.682} C_VEL
LIN {X 0,Y 213.149,Z 590.265,A -85,B 0,C 180,E1 -20606.219,E2 -20606.219} C_VEL
LIN {X 0,Y 214.027,Z 591.263,A -85,B 0,C 180,E1 -20610,E2 -20610} C_VEL
LIN {X 0,Y 213.163,Z 590.25,A -85,B 0,C 180,E1 -20613.781,E2 -20613.781} C_VEL
LIN {X 0,Y 212.561,Z 587.844,A -85,B 0,C 180,E1 -20617.294,E2 -20617.294} C_VEL
LIN {X 0,Y 212.463,Z 584.41,A -85,B 0,C 180,E1 -20620.482,E2 -20620.482} C_VEL
LIN {X 0,Y 212.893,Z 580.198,A -85,B 0,C 180,E1 -20623.361,E2 -20623.361} C_VEL
LIN {X 0,Y 214.162,Z 573.82,A -85,B 0,C 180,E1 -20626.687,E2 -20626.687} C_VEL
LIN {X 0,Y 215.589,Z 568.203,A -85,B 0,C 180,E1 -20629.025,E2 -20629.025} C_VEL
LIN {X 0,Y 217.836,Z 559.975,A -85,B 0,C 180,E1 -20631.778,E2 -20631.778} C_VEL
LIN {X 0,Y 220.243,Z 551.648,A -85,B 0,C 180,E1 -20634.007,E2 -20634.007} C_VEL
LIN {X 0,Y 223.034,Z 541.53,A -85,B 0,C 180,E1 -20636.177,E2 -20636.177} C_VEL
LIN {X 0,Y 226.039,Z 530.151,A -85,B 0,C 180,E1 -20638.051,E2 -20638.051} C_VEL
LIN {X 0,Y 228.532,Z 519.02,A -85,B 0,C 180,E1 -20639.474,E2 -20639.474} C_VEL
LIN {X 0,Y 230.637,Z 506.659,A -85,B 0,C 180,E1 -20640.69,E2 -20640.69} C_VEL
LIN {X 0,Y 232.404,Z 493.342,A -85,B 0,C 180,E1 -20641.589,E2 -20641.589} C_VEL
LIN {X 0,Y 233.384,Z 480.121,A -85,B 0,C 180,E1 -20642.166,E2 -20642.166} C_VEL
LIN {X 0,Y 234.273,Z 456.845,A -85,B 0,C 180,E1 -20642.862,E2 -20642.862} C_VEL
LIN {X 0,Y 232.142,Z 427.754,A -85,B 0,C 180,E1 -20644.237,E2 -20644.237} C_VEL
LIN {X 0,Y 229.034,Z 397.829,A -85,B 0,C 180,E1 -20645.861,E2 -20645.861} C_VEL
LIN {X 0,Y 227.529,Z 387.441,A -85,B 0,C 180,E1 -20646.519,E2 -20646.519} C_VEL
LIN {X 0,Y 222.131,Z 375.264,A -85,B 0,C 180,E1 -20648,E2 -20648} C_VEL
LIN {X 0,Y 221.016,Z 372.246,A -85,B 0,C 180,E1 -20648.461,E2 -20648.461} C_VEL
LIN {X 0,Y 218.604,Z 362.132,A -85,B 0,C 180,E1 -20652.464,E2 -20652.464} C_VEL
LIN {X 0,Y 215.852,Z 352.07,A -85,B 0,C 180,E1 -20656.863,E2 -20656.863} C_VEL
LIN {X 0,Y 213.771,Z 344.917,A -85,B 0,C 180,E1 -20660.357,E2 -20660.357} C_VEL
LIN {X 0,Y 213.76,Z 344.795,A -85,B 0,C 180,E1 -20665.279,E2 -20665.279} C_VEL
LIN {X 0,Y 213.765,Z 344.855,A -85,B 0,C 180,E1 -20668.737,E2 -20668.737} C_VEL
LIN {X 0,Y 213.78,Z 344.828,A -85,B 0,C 180,E1 -20672.597,E2 -20672.597} C_VEL
LIN {X 0,Y 213.804,Z 344.83,A -85,B 0,C 180,E1 -20676.981,E2 -20676.981} C_VEL
LIN {X 0,Y 213.939,Z 344.832,A -85,B 0,C 180,E1 -20682.803,E2 -20682.803} C_VEL
LIN {X 0,Y 213.94,Z 344.813,A -85,B 0,C 180,E1 -20686.706,E2 -20686.706} C_VEL
LIN {X 0,Y 214.133,Z 344.812,A -85,B 0,C 180,E1 -20690.555,E2 -20690.555} C_VEL
LIN {X 0,Y 214.073,Z 344.796,A -85,B 0,C 180,E1 -20694.348,E2 -20694.348} C_VEL
LIN {X 0,Y 214.402,Z 344.775,A -85,B 0,C 180,E1 -20698.122,E2 -20698.122} C_VEL
LIN {X 0,Y 214.507,Z 344.742,A -85,B 0,C 180,E1 -20700,E2 -20700} C_VEL
LIN {X 0,Y 214.402,Z 344.756,A -85,B 0,C 180,E1 -20701.879,E2 -20701.879} C_VEL
LIN {X 0,Y 214.175,Z 344.781,A -85,B 0,C 180,E1 -20707.542,E2 -20707.542} C_VEL
LIN {X 0,Y 213.99,Z 344.829,A -85,B 0,C 180,E1 -20711.365,E2 -20711.365} C_VEL
LIN {X 0,Y 213.898,Z 344.818,A -85,B 0,C 180,E1 -20715.24,E2 -20715.24} C_VEL
LIN {X 0,Y 213.808,Z 344.843,A -85,B 0,C 180,E1 -20719.19,E2 -20719.19} C_VEL
LIN {X 0,Y 213.783,Z 344.852,A -85,B 0,C 180,E1 -20723.235,E2 -20723.235} C_VEL
LIN {X 0,Y 213.782,Z 344.802,A -85,B 0,C 180,E1 -20727.427,E2 -20727.427} C_VEL
LIN {X 0,Y 213.756,Z 344.806,A -85,B 0,C 180,E1 -20731.74,E2 -20731.74} C_VEL
LIN {X 0,Y 213.739,Z 344.843,A -85,B 0,C 180,E1 -20736.29,E2 -20736.29} C_VEL
LIN {X 0,Y 213.695,Z 344.828,A -85,B 0,C 180,E1 -20741.129,E2 -20741.129} C_VEL
LIN {X 0,Y 213.699,Z 344.866,A -85,B 0,C 180,E1 -20743.681,E2 -20743.681} C_VEL
LIN {X 0,Y 213.699,Z 344.829,A -85,B 0,C 180,E1 -20746.346,E2 -20746.346} C_VEL
LIN {X 0,Y 213.762,Z 345.034,A -85,B 0,C 180,E1 -20750.734,E2 -20750.734} C_VEL
LIN {X 0,Y 214.013,Z 346.105,A -85,B 0,C 180,E1 -20751.087,E2 -20751.087} C_VEL
LIN {X 0,Y 215.576,Z 348.778,A -85,B 0,C 180,E1 -20751.568,E2 -20751.568} C_VEL
LIN {X 0,Y 216.694,Z 350.382,A -85,B 0,C 180,E1 -20751.878,E2 -20751.878} C_VEL
LIN {X 0,Y 223.276,Z 360.909,A -85,B 0,C 180,E1 -20753.657,E2 -20753.657} C_VEL
LIN {X 0,Y 231.387,Z 375.544,A -85,B 0,C 180,E1 -20755.722,E2 -20755.722} C_VEL
LIN {X 0,Y 237.07,Z 387.198,A -85,B 0,C 180,E1 -20757.105,E2 -20757.105} C_VEL
LIN {X 0,Y 235.997,Z 428.862,A -85,B 0,C 180,E1 -20758.455,E2 -20758.455} C_VEL
LIN {X 0,Y 235.211,Z 441.881,A -85,B 0,C 180,E1 -20759.191,E2 -20759.191} C_VEL
LIN {X 0,Y 233.954,Z 454.906,A -85,B 0,C 180,E1 -20760.288,E2 -20760.288} C_VEL
LIN {X 0,Y 232.298,Z 466.463,A -85,B 0,C 180,E1 -20761.601,E2 -20761.601} C_VEL
LIN {X 0,Y 230.065,Z 477.621,A -85,B 0,C 180,E1 -20763.22,E2 -20763.22} C_VEL
LIN {X 0,Y 227.916,Z 486.9,A -85,B 0,C 180,E1 -20764.914,E2 -20764.914} C_VEL
LIN {X 0,Y 225.639,Z 496.348,A -85,B 0,C 180,E1 -20767.087,E2 -20767.087} C_VEL
LIN {X 0,Y 223.477,Z 504.088,A -85,B 0,C 180,E1 -20769.281,E2 -20769.281} C_VEL
LIN {X 0,Y 221.176,Z 511.747,A -85,B 0,C 180,E1 -20772,E2 -20772} C_VEL
LIN {X 0,Y 219.012,Z 518.549,A -85,B 0,C 180,E1 -20775.125,E2 -20775.125} C_VEL
LIN {X 0,Y 217.397,Z 523.157,A -85,B 0,C 180,E1 -20777.87,E2 -20777.87} C_VEL
LIN {X 0,Y 215.977,Z 526.701,A -85,B 0,C 180,E1 -20780.636,E2 -20780.636} C_VEL
LIN {X 0,Y 215.288,Z 528.524,A -85,B 0,C 180,E1 -20782.497,E2 -20782.497} C_VEL
LIN {X 0,Y 215.006,Z 529.859,A -85,B 0,C 180,E1 -20784.373,E2 -20784.373} C_VEL
LIN {X 0,Y 214.627,Z 530.832,A -85,B 0,C 180,E1 -20786.245,E2 -20786.245} C_VEL
LIN {X 0,Y 214.556,Z 531.408,A -85,B 0,C 180,E1 -20788.123,E2 -20788.123} C_VEL
LIN {X 0,Y 214.499,Z 531.632,A -85,B 0,C 180,E1 -20790,E2 -20790} C_VEL
LIN {X 0,Y 214.556,Z 531.443,A -85,B 0,C 180,E1 -20791.877,E2 -20791.877} C_VEL
LIN {X 0,Y 214.625,Z 530.888,A -85,B 0,C 180,E1 -20793.755,E2 -20793.755} C_VEL
LIN {X 0,Y 214.999,Z 529.937,A -85,B 0,C 180,E1 -20795.628,E2 -20795.628} C_VEL
LIN {X 0,Y 215.273,Z 528.639,A -85,B 0,C 180,E1 -20797.503,E2 -20797.503} C_VEL
LIN {X 0,Y 216.481,Z 525.801,A -85,B 0,C 180,E1 -20800.285,E2 -20800.285} C_VEL
LIN {X 0,Y 217.957,Z 521.969,A -85,B 0,C 180,E1 -20803.045,E2 -20803.045} C_VEL
LIN {X 0,Y 219.562,Z 516.882,A -85,B 0,C 180,E1 -20805.882,E2 -20805.882} C_VEL
LIN {X 0,Y 221.966,Z 509.634,A -85,B 0,C 180,E1 -20808.937,E2 -20808.937} C_VEL
LIN {X 0,Y 224.368,Z 501.6,A -85,B 0,C 180,E1 -20811.595,E2 -20811.595} C_VEL
LIN {X 0,Y 226.515,Z 493.371,A -85,B 0,C 180,E1 -20813.787,E2 -20813.787} C_VEL
LIN {X 0,Y 228.63,Z 484.329,A -85,B 0,C 180,E1 -20815.734,E2 -20815.734} C_VEL
LIN {X 0,Y 231.283,Z 472.763,A -85,B 0,C 180,E1 -20817.65,E2 -20817.65} C_VEL
LIN {X 0,Y 233.282,Z 460.815,A -85,B 0,C 180,E1 -20819.217,E2 -20819.217} C_VEL
LIN {X 0,Y 234.874,Z 448.197,A -85,B 0,C 180,E1 -20820.439,E2 -20820.439} C_VEL
LIN {X 0,Y 235.795,Z 435.913,A -85,B 0,C 180,E1 -20821.309,E2 -20821.309} C_VEL
LIN {X 0,Y 236.152,Z 422.852,A -85,B 0,C 180,E1 -20821.919,E2 -20821.919} C_VEL
LIN {X 0,Y 237.176,Z 387.371,A -85,B 0,C 180,E1 -20823.019,E2 -20823.019} C_VEL
LIN {X 0,Y 229.934,Z 372.721,A -85,B 0,C 180,E1 -20824.794,E2 -20824.794} C_VEL
LIN {X 0,Y 222.003,Z 358.799,A -85,B 0,C 180,E1 -20826.838,E2 -20826.838} C_VEL
LIN {X 0,Y 217.712,Z 352.138,A -85,B 0,C 180,E1 -20827.995,E2 -20827.995} C_VEL
LIN {X 0,Y 215.882,Z 349.123,A -85,B 0,C 180,E1 -20828.516,E2 -20828.516} C_VEL
LIN {X 0,Y 214.241,Z 346.72,A -85,B 0,C 180,E1 -20828.989,E2 -20828.989} C_VEL
LIN {X 0,Y 213.794,Z 345.233,A -85,B 0,C 180,E1 -20829.34,E2 -20829.34} C_VEL
LIN {X 0,Y 213.75,Z 344.874,A -85,B 0,C 180,E1 -20829.878,E2 -20829.878} C_VEL
LIN {X 0,Y 213.7,Z 344.829,A -85,B 0,C 180,E1 -20833.679,E2 -20833.679} C_VEL
LIN {X 0,Y 213.699,Z 344.866,A -85,B 0,C 180,E1 -20836.345,E2 -20836.345} C_VEL
LIN {X 0,Y 213.701,Z 344.814,A -85,B 0,C 180,E1 -20841.328,E2 -20841.328} C_VEL
LIN {X 0,Y 213.751,Z 344.855,A -85,B 0,C 180,E1 -20846.017,E2 -20846.017} C_VEL
LIN {X 0,Y 213.743,Z 344.788,A -85,B 0,C 180,E1 -20850.448,E2 -20850.448} C_VEL
LIN {X 0,Y 213.747,Z 344.851,A -85,B 0,C 180,E1 -20854.695,E2 -20854.695} C_VEL
LIN {X 0,Y 213.774,Z 344.836,A -85,B 0,C 180,E1 -20858.799,E2 -20858.799} C_VEL
LIN {X 0,Y 213.881,Z 344.841,A -85,B 0,C 180,E1 -20862.798,E2 -20862.798} C_VEL
LIN {X 0,Y 213.92,Z 344.82,A -85,B 0,C 180,E1 -20866.704,E2 -20866.704} C_VEL
LIN {X 0,Y 214.129,Z 344.798,A -85,B 0,C 180,E1 -20870.555,E2 -20870.555} C_VEL
LIN {X 0,Y 214.071,Z 344.812,A -85,B 0,C 180,E1 -20874.348,E2 -20874.348} C_VEL
LIN {X 0,Y 214.401,Z 344.756,A -85,B 0,C 180,E1 -20878.121,E2 -20878.121} C_VEL
LIN {X 0,Y 214.506,Z 344.741,A -85,B 0,C 180,E1 -20880,E2 -20880} C_VEL
LIN {X 0,Y 214.401,Z 344.775,A -85,B 0,C 180,E1 -20881.878,E2 -20881.878} C_VEL
LIN {X 0,Y 214.177,Z 344.789,A -85,B 0,C 180,E1 -20887.542,E2 -20887.542} C_VEL
LIN {X 0,Y 213.99,Z 344.814,A -85,B 0,C 180,E1 -20891.365,E2 -20891.365} C_VEL
LIN {X 0,Y 213.905,Z 344.837,A -85,B 0,C 180,E1 -20895.239,E2 -20895.239} C_VEL
LIN {X 0,Y 213.813,Z 344.815,A -85,B 0,C 180,E1 -20899.19,E2 -20899.19} C_VEL
LIN {X 0,Y 213.795,Z 344.837,A -85,B 0,C 180,E1 -20903.233,E2 -20903.233} C_VEL
LIN {X 0,Y 213.782,Z 344.827,A -85,B 0,C 180,E1 -20907.427,E2 -20907.427} C_VEL
LIN {X 0,Y 213.756,Z 344.861,A -85,B 0,C 180,E1 -20911.74,E2 -20911.74} C_VEL
LIN {X 0,Y 213.739,Z 344.85,A -85,B 0,C 180,E1 -20916.289,E2 -20916.289} C_VEL
LIN {X 0,Y 213.753,Z 344.995,A -85,B 0,C 180,E1 -20919.647,E2 -20919.647} C_VEL
LIN {X 0,Y 216.36,Z 353.912,A -85,B 0,C 180,E1 -20923.897,E2 -20923.897} C_VEL
LIN {X 0,Y 219.089,Z 363.971,A -85,B 0,C 180,E1 -20928.23,E2 -20928.23} C_VEL
LIN {X 0,Y 219.888,Z 367.288,A -85,B 0,C 180,E1 -20929.576,E2 -20929.576} C_VEL
LIN {X 0,Y 220.31,Z 369.81,A -85,B 0,C 180,E1 -20930.341,E2 -20930.341} C_VEL
LIN {X 0,Y 220.827,Z 374.609,A -85,B 0,C 180,E1 -20931.214,E2 -20931.214} C_VEL
LIN {X 0,Y 221.252,Z 380.062,A -85,B 0,C 180,E1 -20931.818,E2 -20931.818} C_VEL
LIN {X 0,Y 221.869,Z 388.039,A -85,B 0,C 180,E1 -20932.386,E2 -20932.386} C_VEL
LIN {X 0,Y 222.857,Z 396.044,A -85,B 0,C 180,E1 -20932.89,E2 -20932.89} C_VEL
LIN {X 0,Y 224.961,Z 414.108,A -85,B 0,C 180,E1 -20933.974,E2 -20933.974} C_VEL
LIN {X 0,Y 227.719,Z 446.525,A -85,B 0,C 180,E1 -20935.667,E2 -20935.667} C_VEL
LIN {X 0,Y 228.32,Z 459.178,A -85,B 0,C 180,E1 -20936.232,E2 -20936.232} C_VEL
LIN {X 0,Y 227.074,Z 485.359,A -85,B 0,C 180,E1 -20937.071,E2 -20937.071} C_VEL
LIN {X 0,Y 225.656,Z 498.98,A -85,B 0,C 180,E1 -20937.835,E2 -20937.835} C_VEL
LIN {X 0,Y 223.648,Z 511.716,A -85,B 0,C 180,E1 -20938.9,E2 -20938.9} C_VEL
LIN {X 0,Y 221.208,Z 523.455,A -85,B 0,C 180,E1 -20940.237,E2 -20940.237} C_VEL
LIN {X 0,Y 218.345,Z 534.807,A -85,B 0,C 180,E1 -20941.918,E2 -20941.918} C_VEL
LIN {X 0,Y 215.468,Z 545.073,A -85,B 0,C 180,E1 -20943.875,E2 -20943.875} C_VEL
LIN {X 0,Y 212.673,Z 554.35,A -85,B 0,C 180,E1 -20946.121,E2 -20946.121} C_VEL
LIN {X 0,Y 209.946,Z 563.448,A -85,B 0,C 180,E1 -20948.909,E2 -20948.909} C_VEL
LIN {X 0,Y 208.502,Z 568.451,A -85,B 0,C 180,E1 -20950.782,E2 -20950.782} C_VEL
LIN {X 0,Y 207.048,Z 573.955,A -85,B 0,C 180,E1 -20953.231,E2 -20953.231} C_VEL
LIN {X 0,Y 205.925,Z 579.274,A -85,B 0,C 180,E1 -20956.178,E2 -20956.178} C_VEL
LIN {X 0,Y 205.414,Z 583.465,A -85,B 0,C 180,E1 -20959.154,E2 -20959.154} C_VEL
LIN {X 0,Y 205.487,Z 587.065,A -85,B 0,C 180,E1 -20962.68,E2 -20962.68} C_VEL
LIN {X 0,Y 206.045,Z 589.275,A -85,B 0,C 180,E1 -20966.088,E2 -20966.088} C_VEL
LIN {X 0,Y 206.982,Z 590.282,A -85,B 0,C 180,E1 -20970,E2 -20970} C_VEL
LIN {X 0,Y 206.075,Z 589.261,A -85,B 0,C 180,E1 -20973.911,E2 -20973.911} C_VEL
LIN {X 0,Y 205.482,Z 587.041,A -85,B 0,C 180,E1 -20977.309,E2 -20977.309} C_VEL
LIN {X 0,Y 205.415,Z 583.411,A -85,B 0,C 180,E1 -20980.846,E2 -20980.846} C_VEL
LIN {X 0,Y 205.917,Z 579.199,A -85,B 0,C 180,E1 -20983.822,E2 -20983.822} C_VEL
LIN {X 0,Y 207.279,Z 572.818,A -85,B 0,C 180,E1 -20987.258,E2 -20987.258} C_VEL
LIN {X 0,Y 209.182,Z 565.937,A -85,B 0,C 180,E1 -20990.143,E2 -20990.143} C_VEL
LIN {X 0,Y 211.669,Z 557.459,A -85,B 0,C 180,E1 -20992.962,E2 -20992.962} C_VEL
LIN {X 0,Y 214.336,Z 548.825,A -85,B 0,C 180,E1 -20995.23,E2 -20995.23} C_VEL
LIN {X 0,Y 217.044,Z 539.382,A -85,B 0,C 180,E1 -20997.217,E2 -20997.217} C_VEL
LIN {X 0,Y 220.161,Z 527.724,A -85,B 0,C 180,E1 -20999.131,E2 -20999.131} C_VEL
LIN {X 0,Y 222.742,Z 516.243,A -85,B 0,C 180,E1 -21000.582,E2 -21000.582} C_VEL
LIN {X 0,Y 224.726,Z 504.401,A -85,B 0,C 180,E1 -21001.721,E2 -21001.721} C_VEL
LIN {X 0,Y 226.511,Z 490.771,A -85,B 0,C 180,E1 -21002.623,E2 -21002.623} C_VEL
LIN {X 0,Y 227.493,Z 477.432,A -85,B 0,C 180,E1 -21003.175,E2 -21003.175} C_VEL
LIN {X 0,Y 228.197,Z 456.145,A -85,B 0,C 180,E1 -21003.841,E2 -21003.841} C_VEL
LIN {X 0,Y 225.987,Z 425.861,A -85,B 0,C 180,E1 -21005.337,E2 -21005.337} C_VEL
LIN {X 0,Y 222.893,Z 396.267,A -85,B 0,C 180,E1 -21007.029,E2 -21007.029} C_VEL
LIN {X 0,Y 222.058,Z 390.453,A -85,B 0,C 180,E1 -21007.414,E2 -21007.414} C_VEL
LIN {X 0,Y 215.821,Z 376.151,A -85,B 0,C 180,E1 -21009.237,E2 -21009.237} C_VEL
LIN {X 0,Y 213.526,Z 371.024,A -85,B 0,C 180,E1 -21010.048,E2 -21010.048} C_VEL
LIN {X 0,Y 211.473,Z 362.592,A -85,B 0,C 180,E1 -21013.566,E2 -21013.566} C_VEL
LIN {X 0,Y 208.981,Z 353.54,A -85,B 0,C 180,E1 -21017.732,E2 -21017.732} C_VEL
LIN {X 0,Y 206.688,Z 345.814,A -85,B 0,C 180,E1 -21021.706,E2 -21021.706} C_VEL
LIN {X 0,Y 206.697,Z 345.663,A -85,B 0,C 180,E1 -21024.688,E2 -21024.688} C_VEL
LIN {X 0,Y 206.692,Z 345.725,A -85,B 0,C 180,E1 -21029.334,E2 -21029.334} C_VEL
LIN {X 0,Y 206.691,Z 345.726,A -85,B 0,C 180,E1 -21033.766,E2 -21033.766} C_VEL
LIN {X 0,Y 206.729,Z 345.695,A -85,B 0,C 180,E1 -21038.04,E2 -21038.04} C_VEL
LIN {X 0,Y 206.869,Z 345.704,A -85,B 0,C 180,E1 -21042.196,E2 -21042.196} C_VEL
LIN {X 0,Y 206.884,Z 345.693,A -85,B 0,C 180,E1 -21046.244,E2 -21046.244} C_VEL
LIN {X 0,Y 207.077,Z 345.692,A -85,B 0,C 180,E1 -21050.23,E2 -21050.23} C_VEL
LIN {X 0,Y 207.037,Z 345.671,A -85,B 0,C 180,E1 -21054.155,E2 -21054.155} C_VEL
LIN {X 0,Y 207.341,Z 345.655,A -85,B 0,C 180,E1 -21058.058,E2 -21058.058} C_VEL
LIN {X 0,Y 207.475,Z 345.617,A -85,B 0,C 180,E1 -21060,E2 -21060} C_VEL
LIN {X 0,Y 207.342,Z 345.636,A -85,B 0,C 180,E1 -21061.943,E2 -21061.943} C_VEL
LIN {X 0,Y 207.12,Z 345.659,A -85,B 0,C 180,E1 -21067.801,E2 -21067.801} C_VEL
LIN {X 0,Y 206.913,Z 345.708,A -85,B 0,C 180,E1 -21071.759,E2 -21071.759} C_VEL
LIN {X 0,Y 206.826,Z 345.702,A -85,B 0,C 180,E1 -21075.774,E2 -21075.774} C_VEL
LIN {X 0,Y 206.725,Z 345.717,A -85,B 0,C 180,E1 -21079.875,E2 -21079.875} C_VEL
LIN {X 0,Y 206.718,Z 345.736,A -85,B 0,C 180,E1 -21084.078,E2 -21084.078} C_VEL
LIN {X 0,Y 206.683,Z 345.672,A -85,B 0,C 180,E1 -21088.428,E2 -21088.428} C_VEL
LIN {X 0,Y 206.691,Z 345.71,A -85,B 0,C 180,E1 -21092.959,E2 -21092.959} C_VEL
LIN {X 0,Y 206.698,Z 345.736,A -85,B 0,C 180,E1 -21095.312,E2 -21095.312} C_VEL
LIN {X 0,Y 206.644,Z 345.695,A -85,B 0,C 180,E1 -21100.255,E2 -21100.255} C_VEL
LIN {X 0,Y 206.628,Z 345.73,A -85,B 0,C 180,E1 -21104.418,E2 -21104.418} C_VEL
LIN {X 0,Y 206.691,Z 345.895,A -85,B 0,C 180,E1 -21109.058,E2 -21109.058} C_VEL
LIN {X 0,Y 206.916,Z 346.832,A -85,B 0,C 180,E1 -21109.444,E2 -21109.444} C_VEL
LIN {X 0,Y 208.374,Z 349.508,A -85,B 0,C 180,E1 -21109.953,E2 -21109.953} C_VEL
LIN {X 0,Y 209.608,Z 351.045,A -85,B 0,C 180,E1 -21110.314,E2 -21110.314} C_VEL
LIN {X 0,Y 217.058,Z 362.821,A -85,B 0,C 180,E1 -21112.473,E2 -21112.473} C_VEL
LIN {X 0,Y 225.179,Z 377.153,A -85,B 0,C 180,E1 -21114.658,E2 -21114.658} C_VEL
LIN {X 0,Y 231.079,Z 389.364,A -85,B 0,C 180,E1 -21116.181,E2 -21116.181} C_VEL
LIN {X 0,Y 229.952,Z 430.738,A -85,B 0,C 180,E1 -21117.575,E2 -21117.575} C_VEL
LIN {X 0,Y 229.111,Z 443.833,A -85,B 0,C 180,E1 -21118.359,E2 -21118.359} C_VEL
LIN {X 0,Y 227.877,Z 455.892,A -85,B 0,C 180,E1 -21119.412,E2 -21119.412} C_VEL
LIN {X 0,Y 226.206,Z 467.058,A -85,B 0,C 180,E1 -21120.7,E2 -21120.7} C_VEL
LIN {X 0,Y 223.813,Z 478.603,A -85,B 0,C 180,E1 -21122.409,E2 -21122.409} C_VEL
LIN {X 0,Y 221.569,Z 487.882,A -85,B 0,C 180,E1 -21124.143,E2 -21124.143} C_VEL
LIN {X 0,Y 219.182,Z 497.329,A -85,B 0,C 180,E1 -21126.372,E2 -21126.372} C_VEL
LIN {X 0,Y 216.917,Z 505.069,A -85,B 0,C 180,E1 -21128.624,E2 -21128.624} C_VEL
LIN {X 0,Y 214.503,Z 512.727,A -85,B 0,C 180,E1 -21131.42,E2 -21131.42} C_VEL
LIN {X 0,Y 212.227,Z 519.528,A -85,B 0,C 180,E1 -21134.638,E2 -21134.638} C_VEL
LIN {X 0,Y 210.531,Z 524.136,A -85,B 0,C 180,E1 -21137.468,E2 -21137.468} C_VEL
LIN {X 0,Y 209.042,Z 527.681,A -85,B 0,C 180,E1 -21140.323,E2 -21140.323} C_VEL
LIN {X 0,Y 208.319,Z 529.503,A -85,B 0,C 180,E1 -21142.245,E2 -21142.245} C_VEL
LIN {X 0,Y 208.011,Z 530.837,A -85,B 0,C 180,E1 -21144.183,E2 -21144.183} C_VEL
LIN {X 0,Y 207.614,Z 531.81,A -85,B 0,C 180,E1 -21146.118,E2 -21146.118} C_VEL
LIN {X 0,Y 207.532,Z 532.387,A -85,B 0,C 180,E1 -21148.059,E2 -21148.059} C_VEL
LIN {X 0,Y 207.471,Z 532.609,A -85,B 0,C 180,E1 -21150,E2 -21150} C_VEL
LIN {X 0,Y 207.532,Z 532.42,A -85,B 0,C 180,E1 -21151.941,E2 -21151.941} C_VEL
LIN {X 0,Y 207.612,Z 531.865,A -85,B 0,C 180,E1 -21153.882,E2 -21153.882} C_VEL
LIN {X 0,Y 208.004,Z 530.915,A -85,B 0,C 180,E1 -21155.818,E2 -21155.818} C_VEL
LIN {X 0,Y 208.303,Z 529.616,A -85,B 0,C 180,E1 -21157.756,E2 -21157.756} C_VEL
LIN {X 0,Y 209.57,Z 526.778,A -85,B 0,C 180,E1 -21160.629,E2 -21160.629} C_VEL
LIN {X 0,Y 211.116,Z 522.945,A -85,B 0,C 180,E1 -21163.475,E2 -21163.475} C_VEL
LIN {X 0,Y 212.811,Z 517.859,A -85,B 0,C 180,E1 -21166.4,E2 -21166.4} C_VEL
LIN {X 0,Y 215.331,Z 510.61,A -85,B 0,C 180,E1 -21169.544,E2 -21169.544} C_VEL
LIN {X 0,Y 217.848,Z 502.576,A -85,B 0,C 180,E1 -21172.276,E2 -21172.276} C_VEL
LIN {X 0,Y 220.101,Z 494.346,A -85,B 0,C 180,E1 -21174.525,E2 -21174.525} C_VEL
LIN {X 0,Y 222.308,Z 485.305,A -85,B 0,C 180,E1 -21176.522,E2 -21176.522} C_VEL
LIN {X 0,Y 225.087,Z 473.736,A -85,B 0,C 180,E1 -21178.479,E2 -21178.479} C_VEL
LIN {X 0,Y 227.174,Z 461.787,A -85,B 0,C 180,E1 -21180.082,E2 -21180.082} C_VEL
LIN {X 0,Y 228.836,Z 449.167,A -85,B 0,C 180,E1 -21181.331,E2 -21181.331} C_VEL
LIN {X 0,Y 229.796,Z 436.811,A -85,B 0,C 180,E1 -21182.229,E2 -21182.229} C_VEL
LIN {X 0,Y 230.198,Z 423.809,A -85,B 0,C 180,E1 -21182.847,E2 -21182.847} C_VEL
LIN {X 0,Y 231.231,Z 389.555,A -85,B 0,C 180,E1 -21183.936,E2 -21183.936} C_VEL
LIN {X 0,Y 224.435,Z 375.847,A -85,B 0,C 180,E1 -21185.689,E2 -21185.689} C_VEL
LIN {X 0,Y 217.083,Z 362.795,A -85,B 0,C 180,E1 -21187.686,E2 -21187.686} C_VEL
LIN {X 0,Y 211.245,Z 353.736,A -85,B 0,C 180,E1 -21189.357,E2 -21189.357} C_VEL
LIN {X 0,Y 208.907,Z 350.074,A -85,B 0,C 180,E1 -21190.067,E2 -21190.067} C_VEL
LIN {X 0,Y 207.124,Z 347.51,A -85,B 0,C 180,E1 -21190.624,E2 -21190.624} C_VEL
LIN {X 0,Y 206.736,Z 346.19,A -85,B 0,C 180,E1 -21190.939,E2 -21190.939} C_VEL
LIN {X 0,Y 206.628,Z 345.755,A -85,B 0,C 180,E1 -21191.558,E2 -21191.558} C_VEL
LIN {X 0,Y 206.628,Z 345.73,A -85,B 0,C 180,E1 -21195.582,E2 -21195.582} C_VEL
LIN {X 0,Y 206.645,Z 345.697,A -85,B 0,C 180,E1 -21199.745,E2 -21199.745} C_VEL
LIN {X 0,Y 206.698,Z 345.735,A -85,B 0,C 180,E1 -21204.688,E2 -21204.688} C_VEL
LIN {X 0,Y 206.691,Z 345.67,A -85,B 0,C 180,E1 -21209.334,E2 -21209.334} C_VEL
LIN {X 0,Y 206.682,Z 345.709,A -85,B 0,C 180,E1 -21213.765,E2 -21213.765} C_VEL
LIN {X 0,Y 206.71,Z 345.719,A -85,B 0,C 180,E1 -21218.038,E2 -21218.038} C_VEL
LIN {X 0,Y 206.819,Z 345.724,A -85,B 0,C 180,E1 -21222.192,E2 -21222.192} C_VEL
LIN {X 0,Y 206.861,Z 345.695,A -85,B 0,C 180,E1 -21226.242,E2 -21226.242} C_VEL
LIN {X 0,Y 207.074,Z 345.68,A -85,B 0,C 180,E1 -21230.23,E2 -21230.23} C_VEL
LIN {X 0,Y 207.034,Z 345.687,A -85,B 0,C 180,E1 -21234.155,E2 -21234.155} C_VEL
LIN {X 0,Y 207.341,Z 345.636,A -85,B 0,C 180,E1 -21238.057,E2 -21238.057} C_VEL
LIN {X 0,Y 207.474,Z 345.617,A -85,B 0,C 180,E1 -21240,E2 -21240} C_VEL
LIN {X 0,Y 207.341,Z 345.654,A -85,B 0,C 180,E1 -21241.942,E2 -21241.942} C_VEL
LIN {X 0,Y 207.122,Z 345.67,A -85,B 0,C 180,E1 -21247.801,E2 -21247.801} C_VEL
LIN {X 0,Y 206.913,Z 345.691,A -85,B 0,C 180,E1 -21251.759,E2 -21251.759} C_VEL
LIN {X 0,Y 206.84,Z 345.72,A -85,B 0,C 180,E1 -21255.773,E2 -21255.773} C_VEL
LIN {X 0,Y 206.854,Z 345.701,A -85,B 0,C 180,E1 -21257.955,E2 -21257.955} C_VEL
LIN {X 0,Y 206.737,Z 345.717,A -85,B 0,C 180,E1 -21263.387,E2 -21263.387} C_VEL
LIN {X 0,Y 206.684,Z 345.707,A -85,B 0,C 180,E1 -21268.428,E2 -21268.428} C_VEL
LIN {X 0,Y 206.691,Z 345.725,A -85,B 0,C 180,E1 -21272.959,E2 -21272.959} C_VEL
LIN {X 0,Y 206.666,Z 345.735,A -85,B 0,C 180,E1 -21277.743,E2 -21277.743} C_VEL
LIN {X 0,Y 206.72,Z 346.008,A -85,B 0,C 180,E1 -21278.367,E2 -21278.367} C_VEL
LIN {X 0,Y 209.382,Z 354.841,A -85,B 0,C 180,E1 -21282.819,E2 -21282.819} C_VEL
LIN {X 0,Y 211.789,Z 363.796,A -85,B 0,C 180,E1 -21286.891,E2 -21286.891} C_VEL
LIN {X 0,Y 213.61,Z 371.182,A -85,B 0,C 180,E1 -21289.938,E2 -21289.938} C_VEL
LIN {X 0,Y 218.732,Z 382.587,A -85,B 0,C 180,E1 -21291.553,E2 -21291.553} C_VEL
LIN {X 0,Y 222.376,Z 391.361,A -85,B 0,C 180,E1 -21292.616,E2 -21292.616} C_VEL
LIN {X 0,Y 222.857,Z 396.044,A -85,B 0,C 180,E1 -21292.89,E2 -21292.89} C_VEL
LIN {X 0,Y 223.141,Z 401.831,A -85,B 0,C 180,E1 -21293.169,E2 -21293.169} C_VEL
LIN {X 0,Y 221.804,Z 411.654,A -85,B 0,C 180,E1 -21293.304,E2 -21293.304} C_VEL
LIN {X 0,Y 220.281,Z 421.527,A -85,B 0,C 180,E1 -21293.407,E2 -21293.407} C_VEL
LIN {X 0,Y 220.296,Z 427.404,A -85,B 0,C 180,E1 -21293.64,E2 -21293.64} C_VEL
LIN {X 0,Y 222.429,Z 457.598,A -85,B 0,C 180,E1 -21295.187,E2 -21295.187} C_VEL
LIN {X 0,Y 221.21,Z 483.482,A -85,B 0,C 180,E1 -21296.028,E2 -21296.028} C_VEL
LIN {X 0,Y 219.88,Z 495.962,A -85,B 0,C 180,E1 -21296.702,E2 -21296.702} C_VEL
LIN {X 0,Y 218.019,Z 508.607,A -85,B 0,C 180,E1 -21297.731,E2 -21297.731} C_VEL
LIN {X 0,Y 215.43,Z 520.876,A -85,B 0,C 180,E1 -21299.082,E2 -21299.082} C_VEL
LIN {X 0,Y 212.483,Z 532.523,A -85,B 0,C 180,E1 -21300.8,E2 -21300.8} C_VEL
LIN {X 0,Y 209.36,Z 543.024,A -85,B 0,C 180,E1 -21302.783,E2 -21302.783} C_VEL
LIN {X 0,Y 206.724,Z 551.661,A -85,B 0,C 180,E1 -21304.852,E2 -21304.852} C_VEL
LIN {X 0,Y 204.168,Z 559.66,A -85,B 0,C 180,E1 -21307.217,E2 -21307.217} C_VEL
LIN {X 0,Y 201.661,Z 567.883,A -85,B 0,C 180,E1 -21310.297,E2 -21310.297} C_VEL
LIN {X 0,Y 200.417,Z 571.922,A -85,B 0,C 180,E1 -21312.132,E2 -21312.132} C_VEL
LIN {X 0,Y 198.968,Z 578.278,A -85,B 0,C 180,E1 -21315.685,E2 -21315.685} C_VEL
LIN {X 0,Y 198.392,Z 582.47,A -85,B 0,C 180,E1 -21318.765,E2 -21318.765} C_VEL
LIN {X 0,Y 198.42,Z 586.243,A -85,B 0,C 180,E1 -21322.637,E2 -21322.637} C_VEL
LIN {X 0,Y 198.945,Z 588.285,A -85,B 0,C 180,E1 -21325.949,E2 -21325.949} C_VEL
LIN {X 0,Y 199.936,Z 589.302,A -85,B 0,C 180,E1 -21330,E2 -21330} C_VEL
LIN {X 0,Y 198.971,Z 588.27,A -85,B 0,C 180,E1 -21334.051,E2 -21334.051} C_VEL
LIN {X 0,Y 198.42,Z 586.21,A -85,B 0,C 180,E1 -21337.362,E2 -21337.362} C_VEL
LIN {X 0,Y 198.392,Z 582.414,A -85,B 0,C 180,E1 -21341.235,E2 -21341.235} C_VEL
LIN {X 0,Y 198.96,Z 578.199,A -85,B 0,C 180,E1 -21344.315,E2 -21344.315} C_VEL
LIN {X 0,Y 200.405,Z 571.813,A -85,B 0,C 180,E1 -21347.869,E2 -21347.869} C_VEL
LIN {X 0,Y 202.479,Z 564.939,A -85,B 0,C 180,E1 -21350.841,E2 -21350.841} C_VEL
LIN {X 0,Y 205.108,Z 556.463,A -85,B 0,C 180,E1 -21353.741,E2 -21353.741} C_VEL
LIN {X 0,Y 207.9,Z 547.829,A -85,B 0,C 180,E1 -21356.069,E2 -21356.069} C_VEL
LIN {X 0,Y 211.032,Z 537.196,A -85,B 0,C 180,E1 -21358.331,E2 -21358.331} C_VEL
LIN {X 0,Y 213.962,Z 526.727,A -85,B 0,C 180,E1 -21360.06,E2 -21360.06} C_VEL
LIN {X 0,Y 216.655,Z 515.249,A -85,B 0,C 180,E1 -21361.538,E2 -21361.538} C_VEL
LIN {X 0,Y 218.713,Z 503.405,A -85,B 0,C 180,E1 -21362.7,E2 -21362.7} C_VEL
LIN {X 0,Y 220.539,Z 489.894,A -85,B 0,C 180,E1 -21363.612,E2 -21363.612} C_VEL
LIN {X 0,Y 221.501,Z 477.534,A -85,B 0,C 180,E1 -21364.147,E2 -21364.147} C_VEL
LIN {X 0,Y 222.259,Z 457.035,A -85,B 0,C 180,E1 -21364.801,E2 -21364.801} C_VEL
LIN {X 0,Y 220.06,Z 425.486,A -85,B 0,C 180,E1 -21366.413,E2 -21366.413} C_VEL
LIN {X 0,Y 216.84,Z 394.579,A -85,B 0,C 180,E1 -21368.27,E2 -21368.27} C_VEL
LIN {X 0,Y 216.147,Z 392.337,A -85,B 0,C 180,E1 -21368.502,E2 -21368.502} C_VEL
LIN {X 0,Y 210.956,Z 380.182,A -85,B 0,C 180,E1 -21370.112,E2 -21370.112} C_VEL
LIN {X 0,Y 206.108,Z 369.903,A -85,B 0,C 180,E1 -21371.745,E2 -21371.745} C_VEL
LIN {X 0,Y 203.82,Z 361.002,A -85,B 0,C 180,E1 -21375.713,E2 -21375.713} C_VEL
LIN {X 0,Y 201.25,Z 352.032,A -85,B 0,C 180,E1 -21380.198,E2 -21380.198} C_VEL
LIN {X 0,Y 199.615,Z 346.7,A -85,B 0,C 180,E1 -21383.235,E2 -21383.235} C_VEL
LIN {X 0,Y 199.682,Z 346.613,A -85,B 0,C 180,E1 -21388.134,E2 -21388.134} C_VEL
LIN {X 0,Y 199.635,Z 346.59,A -85,B 0,C 180,E1 -21392.764,E2 -21392.764} C_VEL
LIN {X 0,Y 199.682,Z 346.582,A -85,B 0,C 180,E1 -21397.222,E2 -21397.222} C_VEL
LIN {X 0,Y 199.793,Z 346.575,A -85,B 0,C 180,E1 -21401.759,E2 -21401.759} C_VEL
LIN {X 0,Y 199.826,Z 346.576,A -85,B 0,C 180,E1 -21405.748,E2 -21405.748} C_VEL
LIN {X 0,Y 200.02,Z 346.569,A -85,B 0,C 180,E1 -21409.882,E2 -21409.882} C_VEL
LIN {X 0,Y 200.001,Z 346.547,A -85,B 0,C 180,E1 -21413.949,E2 -21413.949} C_VEL
LIN {X 0,Y 200.283,Z 346.535,A -85,B 0,C 180,E1 -21417.989,E2 -21417.989} C_VEL
LIN {X 0,Y 200.443,Z 346.492,A -85,B 0,C 180,E1 -21420,E2 -21420} C_VEL
LIN {X 0,Y 199.99,Z 346.574,A -85,B 0,C 180,E1 -21424.03,E2 -21424.03} C_VEL
LIN {X 0,Y 200.069,Z 346.537,A -85,B 0,C 180,E1 -21428.078,E2 -21428.078} C_VEL
LIN {X 0,Y 199.862,Z 346.584,A -85,B 0,C 180,E1 -21432.18,E2 -21432.18} C_VEL
LIN {X 0,Y 199.763,Z 346.588,A -85,B 0,C 180,E1 -21436.347,E2 -21436.347} C_VEL
LIN {X 0,Y 199.653,Z 346.594,A -85,B 0,C 180,E1 -21440.61,E2 -21440.61} C_VEL
LIN {X 0,Y 199.632,Z 346.612,A -85,B 0,C 180,E1 -21444.99,E2 -21444.99} C_VEL
LIN {X 0,Y 199.604,Z 346.547,A -85,B 0,C 180,E1 -21449.534,E2 -21449.534} C_VEL
LIN {X 0,Y 199.662,Z 346.569,A -85,B 0,C 180,E1 -21452.353,E2 -21452.353} C_VEL
LIN {X 0,Y 199.614,Z 346.588,A -85,B 0,C 180,E1 -21456.765,E2 -21456.765} C_VEL
LIN {X 0,Y 199.592,Z 346.568,A -85,B 0,C 180,E1 -21459.332,E2 -21459.332} C_VEL
LIN {X 0,Y 199.563,Z 346.608,A -85,B 0,C 180,E1 -21462.308,E2 -21462.308} C_VEL
LIN {X 0,Y 199.608,Z 346.754,A -85,B 0,C 180,E1 -21467.176,E2 -21467.176} C_VEL
LIN {X 0,Y 199.772,Z 347.615,A -85,B 0,C 180,E1 -21467.628,E2 -21467.628} C_VEL
LIN {X 0,Y 201.225,Z 350.337,A -85,B 0,C 180,E1 -21468.195,E2 -21468.195} C_VEL
LIN {X 0,Y 202.729,Z 352.107,A -85,B 0,C 180,E1 -21468.67,E2 -21468.67} C_VEL
LIN {X 0,Y 210.523,Z 364.162,A -85,B 0,C 180,E1 -21471.101,E2 -21471.101} C_VEL
LIN {X 0,Y 217.737,Z 376.618,A -85,B 0,C 180,E1 -21473.182,E2 -21473.182} C_VEL
LIN {X 0,Y 224.866,Z 390.781,A -85,B 0,C 180,E1 -21475.128,E2 -21475.128} C_VEL
LIN {X 0,Y 225.23,Z 391.583,A -85,B 0,C 180,E1 -21475.225,E2 -21475.225} C_VEL
LIN {X 0,Y 224.064,Z 431.573,A -85,B 0,C 180,E1 -21476.604,E2 -21476.604} C_VEL
LIN {X 0,Y 223.141,Z 444.925,A -85,B 0,C 180,E1 -21477.419,E2 -21477.419} C_VEL
LIN {X 0,Y 221.853,Z 456.878,A -85,B 0,C 180,E1 -21478.488,E2 -21478.488} C_VEL
LIN {X 0,Y 220.105,Z 468.041,A -85,B 0,C 180,E1 -21479.805,E2 -21479.805} C_VEL
LIN {X 0,Y 217.608,Z 479.586,A -85,B 0,C 180,E1 -21481.552,E2 -21481.552} C_VEL
LIN {X 0,Y 215.264,Z 488.863,A -85,B 0,C 180,E1 -21483.327,E2 -21483.327} C_VEL
LIN {X 0,Y 212.76,Z 498.311,A -85,B 0,C 180,E1 -21485.613,E2 -21485.613} C_VEL
LIN {X 0,Y 210.388,Z 506.049,A -85,B 0,C 180,E1 -21487.926,E2 -21487.926} C_VEL
LIN {X 0,Y 207.854,Z 513.707,A -85,B 0,C 180,E1 -21490.803,E2 -21490.803} C_VEL
LIN {X 0,Y 205.459,Z 520.508,A -85,B 0,C 180,E1 -21494.119,E2 -21494.119} C_VEL
LIN {X 0,Y 203.676,Z 525.115,A -85,B 0,C 180,E1 -21497.039,E2 -21497.039} C_VEL
LIN {X 0,Y 202.114,Z 528.66,A -85,B 0,C 180,E1 -21499.988,E2 -21499.988} C_VEL
LIN {X 0,Y 201.354,Z 530.482,A -85,B 0,C 180,E1 -21501.975,E2 -21501.975} C_VEL
LIN {X 0,Y 201.019,Z 531.816,A -85,B 0,C 180,E1 -21503.98,E2 -21503.98} C_VEL
LIN {X 0,Y 200.602,Z 532.789,A -85,B 0,C 180,E1 -21505.982,E2 -21505.982} C_VEL
LIN {X 0,Y 200.508,Z 533.365,A -85,B 0,C 180,E1 -21507.991,E2 -21507.991} C_VEL
LIN {X 0,Y 200.443,Z 533.587,A -85,B 0,C 180,E1 -21510,E2 -21510} C_VEL
LIN {X 0,Y 200.508,Z 533.398,A -85,B 0,C 180,E1 -21512.009,E2 -21512.009} C_VEL
LIN {X 0,Y 200.601,Z 532.843,A -85,B 0,C 180,E1 -21514.018,E2 -21514.018} C_VEL
LIN {X 0,Y 201.012,Z 531.892,A -85,B 0,C 180,E1 -21516.021,E2 -21516.021} C_VEL
LIN {X 0,Y 201.338,Z 530.594,A -85,B 0,C 180,E1 -21518.026,E2 -21518.026} C_VEL
LIN {X 0,Y 202.667,Z 527.755,A -85,B 0,C 180,E1 -21520.995,E2 -21520.995} C_VEL
LIN {X 0,Y 204.288,Z 523.922,A -85,B 0,C 180,E1 -21523.935,E2 -21523.935} C_VEL
LIN {X 0,Y 206.078,Z 518.835,A -85,B 0,C 180,E1 -21526.952,E2 -21526.952} C_VEL
LIN {X 0,Y 208.721,Z 511.586,A -85,B 0,C 180,E1 -21530.19,E2 -21530.19} C_VEL
LIN {X 0,Y 211.36,Z 503.551,A -85,B 0,C 180,E1 -21532.998,E2 -21532.998} C_VEL
LIN {X 0,Y 213.725,Z 495.321,A -85,B 0,C 180,E1 -21535.308,E2 -21535.308} C_VEL
LIN {X 0,Y 216.033,Z 486.28,A -85,B 0,C 180,E1 -21537.355,E2 -21537.355} C_VEL
LIN {X 0,Y 218.682,Z 475.735,A -85,B 0,C 180,E1 -21539.202,E2 -21539.202} C_VEL
LIN {X 0,Y 220.895,Z 464.04,A -85,B 0,C 180,E1 -21540.838,E2 -21540.838} C_VEL
LIN {X 0,Y 222.648,Z 452.548,A -85,B 0,C 180,E1 -21542.051,E2 -21542.051} C_VEL
LIN {X 0,Y 223.716,Z 439.878,A -85,B 0,C 180,E1 -21543.06,E2 -21543.06} C_VEL
LIN {X 0,Y 224.278,Z 426.153,A -85,B 0,C 180,E1 -21543.77,E2 -21543.77} C_VEL
LIN {X 0,Y 225.366,Z 391.8,A -85,B 0,C 180,E1 -21544.896,E2 -21544.896} C_VEL
LIN {X 0,Y 218.403,Z 377.786,A -85,B 0,C 180,E1 -21546.796,E2 -21546.796} C_VEL
LIN {X 0,Y 211.606,Z 365.866,A -85,B 0,C 180,E1 -21548.748,E2 -21548.748} C_VEL
LIN {X 0,Y 206.558,Z 358.041,A -85,B 0,C 180,E1 -21550.274,E2 -21550.274} C_VEL
LIN {X 0,Y 204.292,Z 354.622,A -85,B 0,C 180,E1 -21550.992,E2 -21550.992} C_VEL
LIN {X 0,Y 201.91,Z 351.034,A -85,B 0,C 180,E1 -21551.772,E2 -21551.772} C_VEL
LIN {X 0,Y 200.172,Z 348.673,A -85,B 0,C 180,E1 -21552.351,E2 -21552.351} C_VEL
LIN {X 0,Y 199.652,Z 347.062,A -85,B 0,C 180,E1 -21552.752,E2 -21552.752} C_VEL
LIN {X 0,Y 199.558,Z 346.589,A -85,B 0,C 180,E1 -21553.634,E2 -21553.634} C_VEL
LIN {X 0,Y 199.568,Z 346.604,A -85,B 0,C 180,E1 -21558.002,E2 -21558.002} C_VEL
LIN {X 0,Y 199.594,Z 346.569,A -85,B 0,C 180,E1 -21560.772,E2 -21560.772} C_VEL
LIN {X 0,Y 199.61,Z 346.62,A -85,B 0,C 180,E1 -21565.713,E2 -21565.713} C_VEL
LIN {X 0,Y 199.683,Z 346.558,A -85,B 0,C 180,E1 -21568.134,E2 -21568.134} C_VEL
LIN {X 0,Y 199.631,Z 346.564,A -85,B 0,C 180,E1 -21572.763,E2 -21572.763} C_VEL
LIN {X 0,Y 199.668,Z 346.604,A -85,B 0,C 180,E1 -21577.22,E2 -21577.22} C_VEL
LIN {X 0,Y 199.743,Z 346.604,A -85,B 0,C 180,E1 -21581.802,E2 -21581.802} C_VEL
LIN {X 0,Y 199.798,Z 346.572,A -85,B 0,C 180,E1 -21585.745,E2 -21585.745} C_VEL
LIN {X 0,Y 200.02,Z 346.562,A -85,B 0,C 180,E1 -21589.881,E2 -21589.881} C_VEL
LIN {X 0,Y 199.998,Z 346.559,A -85,B 0,C 180,E1 -21593.948,E2 -21593.948} C_VEL
LIN {X 0,Y 200.283,Z 346.515,A -85,B 0,C 180,E1 -21597.989,E2 -21597.989} C_VEL
LIN {X 0,Y 200.442,Z 346.492,A -85,B 0,C 180,E1 -21600,E2 -21600} C_VEL
LIN {X 0,Y 199.985,Z 346.563,A -85,B 0,C 180,E1 -21604.03,E2 -21604.03} C_VEL
LIN {X 0,Y 200.07,Z 346.552,A -85,B 0,C 180,E1 -21608.077,E2 -21608.077} C_VEL
LIN {X 0,Y 199.863,Z 346.566,A -85,B 0,C 180,E1 -21612.18,E2 -21612.18} C_VEL
LIN {X 0,Y 199.784,Z 346.599,A -85,B 0,C 180,E1 -21616.345,E2 -21616.345} C_VEL
LIN {X 0,Y 199.774,Z 346.572,A -85,B 0,C 180,E1 -21618.458,E2 -21618.458} C_VEL
LIN {X 0,Y 199.7,Z 346.6,A -85,B 0,C 180,E1 -21623.795,E2 -21623.795} C_VEL
LIN {X 0,Y 199.661,Z 346.581,A -85,B 0,C 180,E1 -21628.361,E2 -21628.361} C_VEL
LIN {X 0,Y 199.662,Z 346.608,A -85,B 0,C 180,E1 -21632.353,E2 -21632.353} C_VEL
LIN {X 0,Y 199.615,Z 346.72,A -85,B 0,C 180,E1 -21636.765,E2 -21636.765} C_VEL
LIN {X 0,Y 202.196,Z 355.149,A -85,B 0,C 180,E1 -21641.331,E2 -21641.331} C_VEL
LIN {X 0,Y 204.537,Z 363.706,A -85,B 0,C 180,E1 -21645.478,E2 -21645.478} C_VEL
LIN {X 0,Y 206.113,Z 369.876,A -85,B 0,C 180,E1 -21648.171,E2 -21648.171} C_VEL
LIN {X 0,Y 211.583,Z 381.569,A -85,B 0,C 180,E1 -21650.01,E2 -21650.01} C_VEL
LIN {X 0,Y 216.755,Z 393.633,A -85,B 0,C 180,E1 -21651.604,E2 -21651.604} C_VEL
LIN {X 0,Y 219.233,Z 415.672,A -85,B 0,C 180,E1 -21652.978,E2 -21652.978} C_VEL
LIN {X 0,Y 220.296,Z 427.404,A -85,B 0,C 180,E1 -21653.64,E2 -21653.64} C_VEL
LIN {X 0,Y 220.334,Z 433.224,A -85,B 0,C 180,E1 -21653.875,E2 -21653.875} C_VEL
LIN {X 0,Y 218.786,Z 442.985,A -85,B 0,C 180,E1 -21653.973,E2 -21653.973} C_VEL
LIN {X 0,Y 217.241,Z 450.827,A -85,B 0,C 180,E1 -21653.997,E2 -21653.997} C_VEL
LIN {X 0,Y 216.582,Z 456.735,A -85,B 0,C 180,E1 -21654.109,E2 -21654.109} C_VEL
LIN {X 0,Y 216.547,Z 458.703,A -85,B 0,C 180,E1 -21654.181,E2 -21654.181} C_VEL
LIN {X 0,Y 215.246,Z 483.554,A -85,B 0,C 180,E1 -21655.017,E2 -21655.017} C_VEL
LIN {X 0,Y 213.837,Z 496.057,A -85,B 0,C 180,E1 -21655.732,E2 -21655.732} C_VEL
LIN {X 0,Y 211.831,Z 508.74,A -85,B 0,C 180,E1 -21656.81,E2 -21656.81} C_VEL
LIN {X 0,Y 208.971,Z 521.484,A -85,B 0,C 180,E1 -21658.299,E2 -21658.299} C_VEL
LIN {X 0,Y 205.93,Z 532.839,A -85,B 0,C 180,E1 -21660.058,E2 -21660.058} C_VEL
LIN {X 0,Y 202.718,Z 543.088,A -85,B 0,C 180,E1 -21662.094,E2 -21662.094} C_VEL
LIN {X 0,Y 199.72,Z 552.372,A -85,B 0,C 180,E1 -21664.465,E2 -21664.465} C_VEL
LIN {X 0,Y 196.655,Z 561.459,A -85,B 0,C 180,E1 -21667.408,E2 -21667.408} C_VEL
LIN {X 0,Y 194.561,Z 567.906,A -85,B 0,C 180,E1 -21670.038,E2 -21670.038} C_VEL
LIN {X 0,Y 192.845,Z 573.852,A -85,B 0,C 180,E1 -21673.05,E2 -21673.05} C_VEL
LIN {X 0,Y 191.737,Z 578.787,A -85,B 0,C 180,E1 -21676.217,E2 -21676.217} C_VEL
LIN {X 0,Y 191.275,Z 582.62,A -85,B 0,C 180,E1 -21679.414,E2 -21679.414} C_VEL
LIN {X 0,Y 191.346,Z 585.434,A -85,B 0,C 180,E1 -21682.609,E2 -21682.609} C_VEL
